(* CoDeSys 2.3 library: TcBACnet.lib *)
(* Libraries: standard.lib 5.6.98 12:03:02, TcBase.lib 14.5.09 12:14:08, TcSystem.lib 27.2.12 15:08:36, TcUtilities.lib 2.3.12 19:25:40 *)

(* Global variable list: BACnet_Globals *)
VAR_GLOBAL
(* global linkable BACnet adapter *)
	fbBACnet_Adapter	: FB_BACnet_Adapter;
(* global visible BACnet adapter reference *)
	pBACnet_Adapter		: POINTER TO FB_BACnet_Adapter;
END_VAR
VAR_GLOBAL CONSTANT
	tBACnet_ADSTimeOut		: TIME := t#5s;
END_VAR

(* Data type *)
TYPE E_BACNETACTION:
(
	BACnetAction_direct :=0,
	BACnetAction_reverse :=1
);
END_TYPE

(* Data type *)
TYPE E_BACNETADAPTERSTATUS :
(
	BACnetAdapterStatus_Init			:= 16#0,
	BACnetAdapterStatus_CheckIpAddr		:= 16#1,
	BACnetAdapterStatus_CheckParam		:= 16#2,
	BACnetAdapterStatus_GetGatewayMAC	:= 16#3,
	BACnetAdapterStatus_WaitGatewayMAC	:= 16#4,
	BACnetAdapterStatus_Complete		:= 16#8
);
END_TYPE

(* Data type *)
TYPE E_BACNETBINARYPV:
(
	BACnetBinaryPV_inactive :=0,
	BACnetBinaryPV_active :=1,
	BACnetBinaryPV_NULL := 2
);
END_TYPE

(* Data type *)
TYPE E_BACNETDATATYPES:
(
	BACnetDataType_Null :=0,
	BACnetDataType_Bool :=1,
	BACnetDataType_UnsignedInteger :=2,
	BACnetDataType_SignedInteger :=3,
	BACnetDataType_Real :=4,
	BACnetDataType_Double :=5,
	BACnetDataType_OctetString :=6,
	BACnetDataType_CharacterStringExt :=7,
	BACnetDataType_BitString :=8,
	BACnetDataType_Enumerated :=9,
	BACnetDataType_Date :=10,
	BACnetDataType_Time :=11,
	BACnetDataType_ObjectIdentifier :=12,
	BACnetDataType_DateTime :=14,
	BACnetDataType_ArrayIndex :=15,
	BACnetDataType_CalendarEntry :=16,
	BACnetDataType_ObjectType :=17,
	BACnetDataType_EventTransitionBits :=18,
	BACnetDataType_ActionList :=19,
	BACnetDataType_StatusFlags :=20,
	BACnetDataType_EventState :=21,
	BACnetDataType_Reliability :=22,
	BACnetDataType_Polarity :=23,
	BACnetDataType_EngineeringUnits :=25,
	BACnetDataType_PriorityValue :=26,
	BACnetDataType_LimitEnable :=27,
	BACnetDataType_NotifyType :=29,
	BACnetDataType_TimeStamp :=30,
	BACnetDataType_DeviceObjectPropertyReference :=31,
	BACnetDataType_DeviceStatus :=32,
	BACnetDataType_ServicesSupported :=33,
	BACnetDataType_ObjectTypesSupported :=34,
	BACnetDataType_Segmentation :=35,
	BACnetDataType_VTClass :=36,
	BACnetDataType_VTSession :=37,
	BACnetDataType_SessionKey :=38,
	BACnetDataType_Recipient :=39,
	BACnetDataType_AddressBinding :=40,
	BACnetDataType_COVSubscription :=41,
	BACnetDataType_EventType :=42,
	BACnetDataType_EventParameter :=43,
	BACnetDataType_FileAccessMethod :=44,
	BACnetDataType_ReadAccessSpecification :=45,
	BACnetDataType_ReadAccessResult :=46,
	BACnetDataType_ObjectPropertyReference :=47,
	BACnetDataType_SetpointReference :=48,
	BACnetDataType_Destination :=49,
	BACnetDataType_ProgramState :=50,
	BACnetDataType_ProgramRequest :=51,
	BACnetDataType_ProgramError :=52,
	BACnetDataType_DateRange :=53,
	BACnetDataType_DailySchedule :=54,
	BACnetDataType_SpecialEvent :=55,
	BACnetDataType_ClientCOV :=56,
	BACnetDataType_LogRecord :=57,
	BACnetDataType_LifeSafetyState :=58,
	BACnetDataType_LifeSafetyMode :=59,
	BACnetDataType_SilencedState :=60,
	BACnetDataType_LifeSafetyOperation :=61,
	BACnetDataType_BinaryPV :=62,
	BACnetDataType_DaysOfWeek :=63,
	BACnetDataType_WeekNDay :=64,
	BACnetDataType_TimeValue :=65,
	BACnetDataType_Value :=66,
	BACnetDataType_Address :=67,
	BACnetDataType_PropertyIdentifier :=68,
	BACnetDataType_EnumerationValueType :=69,
	BACnetDataType_BitFieldBit :=70,
	BACnetDataType_LogDatum :=71,
	BACnetDataType_AnyType :=72,
	BACnetDataType_PresentValue :=73,
	BACnetDataType_ContextTag :=74,
	BACnetDataType_ValueChoice :=75,
	BACnetDataType_LogStatus :=76,
	BACnetDataType_RecipientProcess :=77,
	BACnetDataType_SubscribeCOVPropertyRequest :=78,
	BACnetDataType_PropertyReference :=79,
	BACnetDataType_PropertyResult :=80,
	BACnetDataType_DeviceObjectPropertyValue :=81,
	BACnetDataType_COVNotificationRequest :=82,
	BACnetDataType_EventNotificationRequest :=83,
	BACnetDataType_NotificationParameters :=84,
	BACnetDataType_Change_of_Bitstring :=85,
	BACnetDataType_Change_of_State :=86,
	BACnetDataType_Change_of_Value :=87,
	BACnetDataType_Command_failure :=88,
	BACnetDataType_Floating_limit :=89,
	BACnetDataType_Out_of_Range :=90,
	BACnetDataType_PropertyValue :=91,
	BACnetDataType_Complex_Tag :=92,
	BACnetDataType_Change_of_life_safety :=93,
	BACnetDataType_Extended :=94,
	BACnetDataType_Buffer_ready :=95,
	BACnetDataType_Unsigned_range :=96,
	BACnetDataType_PropertyResultValue :=97,
	BACnetDataType_ServiceCOVPropSubscription :=98,
	BACnetDataType_ServiceCOVSubscription :=99,
	BACnetDataType_COVNotification :=100,
	BACnetDataType_AcknowledgeAlarmRequest :=101,
	BACnetDataType_VTOpenRequest :=102,
	BACnetDataType_Prescale :=103,
	BACnetDataType_Scale :=104,
	BACnetDataType_Action :=105,
	BACnetDataType_Error :=106,
	BACnetDataType_ErrorType :=107,
	BACnetDataType_ErrorClass :=108,
	BACnetDataType_ErrorCode :=109,
	BACnetDataType_RejectReason :=110,
	BACnetDataType_AbortReason :=111,
	BACnetDataType_BDTEntry :=112,
	BACnetDataType_IpEntry :=113,
	BACnetDataType_MaskEntry :=114,
	BACnetDataType_UnsignedIntegerArr :=258,
	BACnetDataType_CharacterStringExtArr :=263,
	BACnetDataType_ObjectIdentifierArr :=268,
	BACnetDataType_CalendarEntryArr :=272,
	BACnetDataType_ActionListArr :=275,
	BACnetDataType_PriorityValueArr :=282,
	BACnetDataType_TimeStampArr :=286,
	BACnetDataType_DeviceObjectPropertyReferenceArr :=287,
	BACnetDataType_VTClassArr :=292,
	BACnetDataType_VTSessionArr :=293,
	BACnetDataType_SessionKeyArr :=294,
	BACnetDataType_RecipientArr :=295,
	BACnetDataType_AddressBindingArr :=296,
	BACnetDataType_COVSubscriptionArr :=297,
	BACnetDataType_ReadAccessSpecificationArr :=301,
	BACnetDataType_ReadAccessResultArr :=302,
	BACnetDataType_DestinationArr :=305,
	BACnetDataType_SpecialEventArr :=311,
	BACnetDataType_LogRecordArr :=313,
	BACnetDataType_LifeSafetyStateArr :=314,
	BACnetDataType_TimeValueArr :=321,
	BACnetDataType_UnsignedIntegerList :=514,
	BACnetDataType_CharacterStringExtList :=519,
	BACnetDataType_ReadAccessSpecificationList :=557,
	BACnetDataType_ReadAccessResultList :=558,
	BACnetDataType_SpecialEventList :=567,
	BACnetDataType_LogRecordList :=569,
	BACnetDataType_TimeValueList :=577,
	BACnetDataType_ValueList :=578,
	BACnetDataType_LogDatumList :=583,
	BACnetDataType_PropertyReferenceList :=591,
	BACnetDataType_PropertyResultList :=592,
	BACnetDataType_COVNotificationRequestList :=594,
	BACnetDataType_EventNotificationRequestList :=595,
	BACnetDataType_PropertyValueList :=603,
	BACnetDataType_DailyScheduleList :=1089
);
END_TYPE

(* Data type *)
TYPE E_BACNETDEVICESTATUS:
(
	BACnetDeviceStatus_Operational :=0,
	BACnetDeviceStatus_OperationalReadOnly :=1,
	BACnetDeviceStatus_DownloadRequired :=2,
	BACnetDeviceStatus_DownloadInProgress :=3,
	BACnetDeviceStatus_NonOperational :=4,
	BACnetDeviceStatus_BackupInProgress :=5
);
END_TYPE

(* Data type *)
TYPE E_BACNETEVENTSTATE:
(
	BACnetEventState_state_normal :=0,
	BACnetEventState_fault :=1,
	BACnetEventState_offnormal :=2,
	BACnetEventState_high_limit :=3,
	BACnetEventState_low_limit :=4,
	BACnetEventState_life_safety_alarm :=5
);
END_TYPE

(* Data type *)
TYPE E_BACNETEVENTTRANSITIONBIT:
(
	BACnetEventTransitionBit_to_offnormal :=0,
	BACnetEventTransitionBit_to_fault :=1,
	BACnetEventTransitionBit_to_normal :=2
);
END_TYPE

(* Data type *)
TYPE E_BACNETEVENTTYPE:
(
	BACnetEventType_change_of_bitstring :=0,
	BACnetEventType_change_of_state :=1,
	BACnetEventType_change_of_value :=2,
	BACnetEventType_command_failure :=3,
	BACnetEventType_floating_limit :=4,
	BACnetEventType_out_of_range :=5,
	BACnetEventType_complex_event_type :=6,
	BACnetEventType_deprecated :=7,
	BACnetEventType_change_of_life_safety :=8,
	BACnetEventType_enumeration :=9,
	BACnetEventType_buffer_ready :=10,
	BACnetEventType_unsigned_range :=11
);
END_TYPE

(* Data type *)
TYPE E_BACNETFILEACCESSMETHOD:
(
	BACnetFileAccessMethod_record_access :=0,
	BACnetFileAccessMethod_stream_access :=1
);
END_TYPE

(* Data type *)
TYPE E_BACNETLIFESAFETYMODE:
(
	BACnetLifeSafetyMode_off :=0,
	BACnetLifeSafetyMode_on :=1,
	BACnetLifeSafetyMode_test :=2,
	BACnetLifeSafetyMode_manned :=3,
	BACnetLifeSafetyMode_unmanned :=4,
	BACnetLifeSafetyMode_armed :=5,
	BACnetLifeSafetyMode_disarmed :=6,
	BACnetLifeSafetyMode_prearmed :=7,
	BACnetLifeSafetyMode_slow :=8,
	BACnetLifeSafetyMode_fast :=9,
	BACnetLifeSafetyMode_disconnected :=10,
	BACnetLifeSafetyMode_enabled :=11,
	BACnetLifeSafetyMode_disabled :=12,
	BACnetLifeSafetyMode_automatic_release_disabled :=13,
	BACnetLifeSafetyMode_mode_default :=14
);
END_TYPE

(* Data type *)
TYPE E_BACNETLIFESAFETYOPERATION:
(
	BACnetLifeSafetyOperation_none :=0,
	BACnetLifeSafetyOperation_silence :=1,
	BACnetLifeSafetyOperation_silence_audible :=2,
	BACnetLifeSafetyOperation_silence_visual :=3,
	BACnetLifeSafetyOperation_reset :=4,
	BACnetLifeSafetyOperation_reset_alarm :=5,
	BACnetLifeSafetyOperation_reset_fault :=6
);
END_TYPE

(* Data type *)
TYPE E_BACNETLIMITENABLEBITS:
(
	BACnetLimitEnableBits_lowLimit :=0,
	BACnetLimitEnableBits_highLimit :=1
);
END_TYPE

(* Data type *)
TYPE E_BACNETNOTIFYTYPE:
(
	BACnetNotifyType_alarm :=0,
	BACnetNotifyType_notify_event :=1,
	BACnetNotifyType_ack_notification :=2
);
END_TYPE

(* Data type *)
TYPE E_BACNETOBJECTSUPPORTEDBITS:
(
	BACnetObjectSupportedBits_AnalogInput :=0,
	BACnetObjectSupportedBits_AnalogOutput :=1,
	BACnetObjectSupportedBits_AnalogValue :=2,
	BACnetObjectSupportedBits_BinaryInput :=3,
	BACnetObjectSupportedBits_BinaryOutput :=4,
	BACnetObjectSupportedBits_BinaryValue :=5,
	BACnetObjectSupportedBits_Calendar :=6,
	BACnetObjectSupportedBits_Command :=7,
	BACnetObjectSupportedBits_Device :=8,
	BACnetObjectSupportedBits_EventEnrollment :=9,
	BACnetObjectSupportedBits_File :=10,
	BACnetObjectSupportedBits_Group :=11,
	BACnetObjectSupportedBits_Loop :=12,
	BACnetObjectSupportedBits_MultiStateInput :=13,
	BACnetObjectSupportedBits_MultiStateOutput :=14,
	BACnetObjectSupportedBits_NotificationClass :=15,
	BACnetObjectSupportedBits_Program :=16,
	BACnetObjectSupportedBits_Schedule :=17,
	BACnetObjectSupportedBits_Averaging :=18,
	BACnetObjectSupportedBits_MultiStateValue :=19,
	BACnetObjectSupportedBits_TrendLog :=20,
	BACnetObjectSupportedBits_LifeSafetyPoint :=21,
	BACnetObjectSupportedBits_LifeSafetyZone :=22
);
END_TYPE

(* Data type *)
TYPE E_BACNETOBJECTTYPE:
(
	BACnetObjectType_AnalogInput :=0,
	BACnetObjectType_AnalogOutput :=1,
	BACnetObjectType_AnalogValue :=2,
	BACnetObjectType_BinaryInput :=3,
	BACnetObjectType_BinaryOutput :=4,
	BACnetObjectType_BinaryValue :=5,
	BACnetObjectType_Calendar :=6,
	BACnetObjectType_Command :=7,
	BACnetObjectType_Device :=8,
	BACnetObjectType_EventEnrollment :=9,
	BACnetObjectType_File :=10,
	BACnetObjectType_Group :=11,
	BACnetObjectType_Loop :=12,
	BACnetObjectType_MultiStateInput :=13,
	BACnetObjectType_MultiStateOutput :=14,
	BACnetObjectType_NotificationClass :=15,
	BACnetObjectType_Program :=16,
	BACnetObjectType_Schedule :=17,
	BACnetObjectType_Averaging :=18,
	BACnetObjectType_MultiStateValue :=19,
	BACnetObjectType_TrendLog :=20,
	BACnetObjectType_LifeSafetyPoint :=21,
	BACnetObjectType_LifeSafetyZone :=22,
	BACnetObjectType_Accumulator :=23,
	BACnetObjectType_PulseConverter :=24,

	(* keep at the end of list! *)
	BACnetObjectType_ZCount
);
END_TYPE

(* Data type *)
TYPE E_BACNETPOLARITY:
(
	BACnetPolarity_normal :=0,
	BACnetPolarity_reverse :=1
);
END_TYPE

(* Data type *)
TYPE E_BACNETPRIORITY:
(
	BACnetPriority_None :=0,
	BACnetPriority_1 :=1,
	BACnetPriority_2 :=2,
	BACnetPriority_3 :=3,
	BACnetPriority_4 :=4,
	BACnetPriority_5 :=5,
	BACnetPriority_6 :=6,
	BACnetPriority_7 :=7,
	BACnetPriority_8 :=8,
	BACnetPriority_9 :=9,
	BACnetPriority_10 :=10,
	BACnetPriority_11 :=11,
	BACnetPriority_12 :=12,
	BACnetPriority_13 :=13,
	BACnetPriority_14 :=14,
	BACnetPriority_15 :=15,
	BACnetPriority_16 :=16
);
END_TYPE

(* Data type *)
TYPE E_BACNETPROGRAMERROR:
(
	BACnetProgramError_program_normal :=0,
	BACnetProgramError_load_failed :=1,
	BACnetProgramError_progerror_internal :=2,
	BACnetProgramError_program :=3,
	BACnetProgramError_other :=4
);
END_TYPE

(* Data type *)
TYPE E_BACNETPROGRAMREQUEST:
(
	BACnetProgramRequest_ready :=0,
	BACnetProgramRequest_load :=1,
	BACnetProgramRequest_run :=2,
	BACnetProgramRequest_halt :=3,
	BACnetProgramRequest_restart :=4,
	BACnetProgramRequest_unload :=5
);
END_TYPE

(* Data type *)
TYPE E_BACNETPROGRAMSTATE:
(
	BACnetProgramState_idle :=0,
	BACnetProgramState_loading :=1,
	BACnetProgramState_running :=2,
	BACnetProgramState_waiting :=3,
	BACnetProgramState_halted :=4,
	BACnetProgramState_unloading :=5
);
END_TYPE

(* Data type *)
TYPE E_BACNETPROPERTYIDENTIFIER:
(
	BACnetPropertyIdentifier_AckedTransitions :=0,
	BACnetPropertyIdentifier_AckRequired :=1,
	BACnetPropertyIdentifier_Action :=2,
	BACnetPropertyIdentifier_ActionText :=3,
	BACnetPropertyIdentifier_ActiveText :=4,
	BACnetPropertyIdentifier_ActiveVtSessions :=5,
	BACnetPropertyIdentifier_AlarmValue :=6,
	BACnetPropertyIdentifier_AlarmValues :=7,
	BACnetPropertyIdentifier_All :=8,
	BACnetPropertyIdentifier_AllWritesSuccessful :=9,
	BACnetPropertyIdentifier_ApduSegmentTimeout :=10,
	BACnetPropertyIdentifier_ApduTimeout :=11,
	BACnetPropertyIdentifier_ApplicationSoftwareVersion :=12,
	BACnetPropertyIdentifier_Archive :=13,
	BACnetPropertyIdentifier_Bias :=14,
	BACnetPropertyIdentifier_ChangeOfStateCount :=15,
	BACnetPropertyIdentifier_ChangeOfStateTime :=16,
	BACnetPropertyIdentifier_NotificationClass :=17,
	BACnetPropertyIdentifier_ControlledVariableReference :=19,
	BACnetPropertyIdentifier_ControlledVariableUnits :=20,
	BACnetPropertyIdentifier_ControlledVariableValue :=21,
	BACnetPropertyIdentifier_CovIncrement :=22,
	BACnetPropertyIdentifier_Datelist :=23,
	BACnetPropertyIdentifier_DaylightSavingsStatus :=24,
	BACnetPropertyIdentifier_Deadband :=25,
	BACnetPropertyIdentifier_DerivativeConstant :=26,
	BACnetPropertyIdentifier_DerivativeConstantUnits :=27,
	BACnetPropertyIdentifier_Description :=28,
	BACnetPropertyIdentifier_DescriptionOfHalt :=29,
	BACnetPropertyIdentifier_DeviceAddressBinding :=30,
	BACnetPropertyIdentifier_DeviceType :=31,
	BACnetPropertyIdentifier_EffectivePeriod :=32,
	BACnetPropertyIdentifier_ElapsedActiveTime :=33,
	BACnetPropertyIdentifier_ErrorLimit :=34,
	BACnetPropertyIdentifier_EventEnable :=35,
	BACnetPropertyIdentifier_EventState :=36,
	BACnetPropertyIdentifier_EventType :=37,
	BACnetPropertyIdentifier_ExceptionSchedule :=38,
	BACnetPropertyIdentifier_FaultValues :=39,
	BACnetPropertyIdentifier_FeedbackValue :=40,
	BACnetPropertyIdentifier_FileAccessMethod :=41,
	BACnetPropertyIdentifier_FileSize :=42,
	BACnetPropertyIdentifier_FileType :=43,
	BACnetPropertyIdentifier_FirmwareRevision :=44,
	BACnetPropertyIdentifier_HighLimit :=45,
	BACnetPropertyIdentifier_InactiveText :=46,
	BACnetPropertyIdentifier_InProcess :=47,
	BACnetPropertyIdentifier_InstanceOf :=48,
	BACnetPropertyIdentifier_IntegralConstant :=49,
	BACnetPropertyIdentifier_IntegralConstantUnits :=50,
	BACnetPropertyIdentifier_IssueConfirmedNotifications :=51,
	BACnetPropertyIdentifier_LimitEnable :=52,
	BACnetPropertyIdentifier_ListOfGroupMembers :=53,
	BACnetPropertyIdentifier_ListOfObjectPropertyReferences :=54,
	BACnetPropertyIdentifier_ListOfSessionKeys :=55,
	BACnetPropertyIdentifier_LocalDate :=56,
	BACnetPropertyIdentifier_LocalTime :=57,
	BACnetPropertyIdentifier_Location :=58,
	BACnetPropertyIdentifier_LowLimit :=59,
	BACnetPropertyIdentifier_ManipulatedVariableReference :=60,
	BACnetPropertyIdentifier_MaximumOutput :=61,
	BACnetPropertyIdentifier_MaxApduLengthAccepted :=62,
	BACnetPropertyIdentifier_MaxInfoFrames :=63,
	BACnetPropertyIdentifier_MaxMaster :=64,
	BACnetPropertyIdentifier_MaxPresValue :=65,
	BACnetPropertyIdentifier_MinimumOfftime :=66,
	BACnetPropertyIdentifier_MinimumOntime :=67,
	BACnetPropertyIdentifier_MinimumOutput :=68,
	BACnetPropertyIdentifier_MinPresValue :=69,
	BACnetPropertyIdentifier_ModelName :=70,
	BACnetPropertyIdentifier_ModificationDate :=71,
	BACnetPropertyIdentifier_NotifyType :=72,
	BACnetPropertyIdentifier_NumberOfAPDURetries :=73,
	BACnetPropertyIdentifier_NumberOfStates :=74,
	BACnetPropertyIdentifier_ObjectIdentifier :=75,
	BACnetPropertyIdentifier_ObjectList :=76,
	BACnetPropertyIdentifier_ObjectName :=77,
	BACnetPropertyIdentifier_ObjectReference :=78,
	BACnetPropertyIdentifier_ObjectType :=79,
	BACnetPropertyIdentifier_Optional :=80,
	BACnetPropertyIdentifier_OutOfService :=81,
	BACnetPropertyIdentifier_OutputUnits :=82,
	BACnetPropertyIdentifier_EventParameters :=83,
	BACnetPropertyIdentifier_Polarity :=84,
	BACnetPropertyIdentifier_PresentValue :=85,
	BACnetPropertyIdentifier_Priority :=86,
	BACnetPropertyIdentifier_PriorityArray :=87,
	BACnetPropertyIdentifier_PriorityForWriting :=88,
	BACnetPropertyIdentifier_ProcessIdentifier :=89,
	BACnetPropertyIdentifier_ProgramChange :=90,
	BACnetPropertyIdentifier_ProgramLocation :=91,
	BACnetPropertyIdentifier_ProgramState :=92,
	BACnetPropertyIdentifier_ProportionalConstant :=93,
	BACnetPropertyIdentifier_ProportionalConstantUnits :=94,
	BACnetPropertyIdentifier_ProtocolObjectTypesSupported :=96,
	BACnetPropertyIdentifier_ProtocolServicesSupported :=97,
	BACnetPropertyIdentifier_ProtocolVersion :=98,
	BACnetPropertyIdentifier_ReadOnly :=99,
	BACnetPropertyIdentifier_ReasonForHalt :=100,
	BACnetPropertyIdentifier_Recipient :=101,
	BACnetPropertyIdentifier_RecipientList :=102,
	BACnetPropertyIdentifier_Reliability :=103,
	BACnetPropertyIdentifier_RelinquishDefault :=104,
	BACnetPropertyIdentifier_Required :=105,
	BACnetPropertyIdentifier_Resolution :=106,
	BACnetPropertyIdentifier_SegmentationSupported :=107,
	BACnetPropertyIdentifier_Setpoint :=108,
	BACnetPropertyIdentifier_SetpointReference :=109,
	BACnetPropertyIdentifier_StateText :=110,
	BACnetPropertyIdentifier_StatusFlags :=111,
	BACnetPropertyIdentifier_SystemStatus :=112,
	BACnetPropertyIdentifier_TimeDelay :=113,
	BACnetPropertyIdentifier_TimeOfActiveTimeReset :=114,
	BACnetPropertyIdentifier_TimeOfStateCountReset :=115,
	BACnetPropertyIdentifier_TimeSynchronizationRecipients :=116,
	BACnetPropertyIdentifier_Units :=117,
	BACnetPropertyIdentifier_UpdateInterval :=118,
	BACnetPropertyIdentifier_UtcOffset :=119,
	BACnetPropertyIdentifier_VendorIdentifier :=120,
	BACnetPropertyIdentifier_VendorName :=121,
	BACnetPropertyIdentifier_VtClassesSupported :=122,
	BACnetPropertyIdentifier_WeeklySchedule :=123,
	BACnetPropertyIdentifier_AttemptedSamples :=124,
	BACnetPropertyIdentifier_AverageValue :=125,
	BACnetPropertyIdentifier_BufferSize :=126,
	BACnetPropertyIdentifier_ClientCovIncrement :=127,
	BACnetPropertyIdentifier_CovResubscriptionInterval :=128,
	BACnetPropertyIdentifier_EventTimeStamps :=130,
	BACnetPropertyIdentifier_LogBuffer :=131,
	BACnetPropertyIdentifier_LogDeviceObjectProperty :=132,
	BACnetPropertyIdentifier_LogEnable :=133,
	BACnetPropertyIdentifier_LogInterval :=134,
	BACnetPropertyIdentifier_MaximumValue :=135,
	BACnetPropertyIdentifier_MinimumValue :=136,
	BACnetPropertyIdentifier_NotificationThreshold :=137,
	BACnetPropertyIdentifier_ProtocolRevision :=139,
	BACnetPropertyIdentifier_RecordsSinceNotification :=140,
	BACnetPropertyIdentifier_RecordCount :=141,
	BACnetPropertyIdentifier_StartTime :=142,
	BACnetPropertyIdentifier_StopTime :=143,
	BACnetPropertyIdentifier_StopWhenFull :=144,
	BACnetPropertyIdentifier_TotalRecordCount :=145,
	BACnetPropertyIdentifier_ValidSamples :=146,
	BACnetPropertyIdentifier_WindowInterval :=147,
	BACnetPropertyIdentifier_WindowSamples :=148,
	BACnetPropertyIdentifier_MaximumValueTimestamp :=149,
	BACnetPropertyIdentifier_MinimumValueTimestamp :=150,
	BACnetPropertyIdentifier_VarianceValue :=151,
	BACnetPropertyIdentifier_ActiveCovSubscriptions :=152,
	BACnetPropertyIdentifier_BackupFailureTimeout :=153,
	BACnetPropertyIdentifier_ConfigurationFiles :=154,
	BACnetPropertyIdentifier_DatabaseRevision :=155,
	BACnetPropertyIdentifier_DirectReading :=156,
	BACnetPropertyIdentifier_LastRestoreTime :=157,
	BACnetPropertyIdentifier_MaintenanceRequired :=158,
	BACnetPropertyIdentifier_MemberOf :=159,
	BACnetPropertyIdentifier_Mode :=160,
	BACnetPropertyIdentifier_OperationExpected :=161,
	BACnetPropertyIdentifier_Setting :=162,
	BACnetPropertyIdentifier_Silenced :=163,
	BACnetPropertyIdentifier_TrackingValue :=164,
	BACnetPropertyIdentifier_ZoneMembers :=165,
	BACnetPropertyIdentifier_LifeSafetyAlarmValues :=166,
	BACnetPropertyIdentifier_MaxSegmentsAccepted :=167,
	BACnetPropertyIdentifier_ProfileName :=168,
	BACnetPropertyIdentifier_InternalUse :=169,
	BACnetPropertyIdentifier_LastNotifyRecord :=173,
	BACnetPropertyIdentifier_ScheduleDefault :=174,
	BACnetPropertyIdentifier_AcceptedModes :=175,
	BACnetPropertyIdentifier_AdjustValue :=176,
	BACnetPropertyIdentifier_Count :=177,
	BACnetPropertyIdentifier_CountBeforeChange :=178,
	BACnetPropertyIdentifier_CovPeriod :=180,
	BACnetPropertyIdentifier_InputReference :=181,
	BACnetPropertyIdentifier_LimitMonitoringInverval :=182,
	BACnetPropertyIdentifier_LoggingObject :=183,
	BACnetPropertyIdentifier_LoggingRecord :=184,
	BACnetPropertyIdentifier_Prescale :=185,
	BACnetPropertyIdentifier_PulseRate :=186,
	BACnetPropertyIdentifier_Scale :=187,
	BACnetPropertyIdentifier_ScaleFactor :=188,
	BACnetPropertyIdentifier_UpdateTime :=189,
	BACnetPropertyIdentifier_ValueBeforeChange :=190,
	BACnetPropertyIdentifier_ValueSet :=191,
	BACnetPropertyIdentifier_ValueChangeTime :=192
);
END_TYPE

(* Data type *)
TYPE E_BACNETRELIABILITY:
(
	BACnetReliability_no_fault_detected :=0,
	BACnetReliability_no_sensor :=1,
	BACnetReliability_over_range :=2,
	BACnetReliability_under_range :=3,
	BACnetReliability_open_loop :=4,
	BACnetReliability_shorted_loop :=5,
	BACnetReliability_no_output :=6,
	BACnetReliability_unreliable_other :=7,
	BACnetReliability_process_error :=8,
	BACnetReliability_multi_state_fault :=9,
	BACnetReliability_configuration_error :=10,
	BACnetReliability_member_fault :=11,
	BACnetReliability_communication_error :=12
);
END_TYPE

(* Data type *)
TYPE E_BACNETSEGMENTATION:
(
	BACnetSegmentation_both :=0,
	BACnetSegmentation_transmit :=1,
	BACnetSegmentation_receive :=2,
	BACnetSegmentation_no :=3
);
END_TYPE

(* Data type *)
TYPE E_BACNETSERVICESUPPORTEDBITS:
(
	BACnetServiceSupportedBits_AcknowledgeAlarm :=0,
	BACnetServiceSupportedBits_ConfirmedCOVNotification :=1,
	BACnetServiceSupportedBits_ConfirmedEventNotification :=2,
	BACnetServiceSupportedBits_GetAlarmSummary :=3,
	BACnetServiceSupportedBits_GetEnrollmentSummary :=4,
	BACnetServiceSupportedBits_SubscribeCOV :=5,
	BACnetServiceSupportedBits_AtomicReadFile :=6,
	BACnetServiceSupportedBits_AtomicWriteFile :=7,
	BACnetServiceSupportedBits_AddListElement :=8,
	BACnetServiceSupportedBits_RemoveListElement :=9,
	BACnetServiceSupportedBits_CreateObject :=10,
	BACnetServiceSupportedBits_DeleteObject :=11,
	BACnetServiceSupportedBits_ReadProperty :=12,
	BACnetServiceSupportedBits_ReadPropertyConditional :=13,
	BACnetServiceSupportedBits_ReadPropertyMultiple :=14,
	BACnetServiceSupportedBits_WriteProperty :=15,
	BACnetServiceSupportedBits_WritePropertyMultiple :=16,
	BACnetServiceSupportedBits_DeviceCommunicationControl :=17,
	BACnetServiceSupportedBits_ConfirmedPrivateTransfer :=18,
	BACnetServiceSupportedBits_ConfirmedTextMessage :=19,
	BACnetServiceSupportedBits_ReinitializeDevice :=20,
	BACnetServiceSupportedBits_VtOpen :=21,
	BACnetServiceSupportedBits_VtClose :=22,
	BACnetServiceSupportedBits_VtData :=23,
	BACnetServiceSupportedBits_Authenticate :=24,
	BACnetServiceSupportedBits_RequestKey :=25,
	BACnetServiceSupportedBits_IAm :=26,
	BACnetServiceSupportedBits_IHave :=27,
	BACnetServiceSupportedBits_UnconfirmedCOVNotification :=28,
	BACnetServiceSupportedBits_UnconfirmedEventNotification :=29,
	BACnetServiceSupportedBits_UnconfirmedPrivateTransfer :=30,
	BACnetServiceSupportedBits_UnconfirmedTextMessage :=31,
	BACnetServiceSupportedBits_TimeSynchronization :=32,
	BACnetServiceSupportedBits_WhoHas :=33,
	BACnetServiceSupportedBits_WhoIs :=34,
	BACnetServiceSupportedBits_ReadRange :=35,
	BACnetServiceSupportedBits_UtcTimeSynchronization :=36,
	BACnetServiceSupportedBits_LifeSafetyOperation :=37,
	BACnetServiceSupportedBits_SubscribeCOVProperty :=38,
	BACnetServiceSupportedBits_GetEventInformation :=39
);
END_TYPE

(* Data type *)
TYPE E_BACNETSILENCEDSTATE:
(
	BACnetSilencedState_unsilenced :=0,
	BACnetSilencedState_audible_silenced :=1,
	BACnetSilencedState_visible_silenced :=2,
	BACnetSilencedState_all_silenced :=3
);
END_TYPE

(* Data type *)
TYPE E_BACNETSTATUSFLAGS:
(
	BACnetStatusFlags_in_alarm :=0,
	BACnetStatusFlags_fault :=1,
	BACnetStatusFlags_overridden :=2,
	BACnetStatusFlags_out_of_service :=3
);
END_TYPE

(* Data type *)
TYPE E_BACNETUNIT:
(
	BACnetUnit_Area_square_meters :=0,
	BACnetUnit_Area_square_feet :=1,
	BACnetUnit_Electrical_milliamperes :=2,
	BACnetUnit_Electrical_amperes :=3,
	BACnetUnit_Electrical_ohms :=4,
	BACnetUnit_Electrical_volts :=5,
	BACnetUnit_Electrical_kilovolts :=6,
	BACnetUnit_Electrical_megavolts :=7,
	BACnetUnit_Electrical_volt_amperes :=8,
	BACnetUnit_Electrical_kilovolt_amperes :=9,
	BACnetUnit_Electrical_megavolt_amperes :=10,
	BACnetUnit_Electrical_volt_amperes_reactive :=11,
	BACnetUnit_Electrical_kilovolt_amperes_reactive :=12,
	BACnetUnit_Electrical_megavolt_amperes_reactive :=13,
	BACnetUnit_Electrical_degrees_phase :=14,
	BACnetUnit_Electrical_power_factor :=15,
	BACnetUnit_Energy_joules :=16,
	BACnetUnit_Energy_kilojoules :=17,
	BACnetUnit_Energy_watt_hours :=18,
	BACnetUnit_Energy_kilowatt_hours :=19,
	BACnetUnit_Energy_btus :=20,
	BACnetUnit_Energy_therms :=21,
	BACnetUnit_Energy_ton_hours :=22,
	BACnetUnit_Enthalpy_joules_per_kilogram_dry_air :=23,
	BACnetUnit_Enthalpy_btus_per_pound_dry_air :=24,
	BACnetUnit_Frequency_cycles_per_hour :=25,
	BACnetUnit_Frequency_cycles_per_minute :=26,
	BACnetUnit_Frequency_hertz :=27,
	BACnetUnit_Humidity_grams_of_water_per_kilogram_dry_air :=28,
	BACnetUnit_Humidity_percent_relative_humidity :=29,
	BACnetUnit_Length_millimeters :=30,
	BACnetUnit_Length_meters :=31,
	BACnetUnit_Length_inches :=32,
	BACnetUnit_Length_feet :=33,
	BACnetUnit_Light_watts_per_square_foot :=34,
	BACnetUnit_Light_watts_per_square_meter :=35,
	BACnetUnit_Light_lumens :=36,
	BACnetUnit_Light_luxes :=37,
	BACnetUnit_Light_foot_candles :=38,
	BACnetUnit_Mass_kilograms :=39,
	BACnetUnit_Mass_pounds_mass :=40,
	BACnetUnit_Mass_tons :=41,
	BACnetUnit_Mass_Flow_kilograms_per_second :=42,
	BACnetUnit_Mass_Flow_kilograms_per_minute :=43,
	BACnetUnit_Mass_Flow_kilograms_per_hour :=44,
	BACnetUnit_Mass_Flow_pounds_mass_per_minute :=45,
	BACnetUnit_Mass_Flow_pounds_mass_per_hour :=46,
	BACnetUnit_Power_watts :=47,
	BACnetUnit_Power_kilowatts :=48,
	BACnetUnit_Power_megawatts :=49,
	BACnetUnit_Power_btus_per_hour :=50,
	BACnetUnit_Power_horsepower :=51,
	BACnetUnit_Power_tons_refrigeration :=52,
	BACnetUnit_Pressure_pascals :=53,
	BACnetUnit_Pressure_kilopascals :=54,
	BACnetUnit_Pressure_bars :=55,
	BACnetUnit_Pressure_pounds_force_per_square_inch :=56,
	BACnetUnit_Pressure_centimeters_of_water :=57,
	BACnetUnit_Pressure_inches_of_water :=58,
	BACnetUnit_Pressure_millimeters_of_mercury :=59,
	BACnetUnit_Pressure_centimeters_of_mercury :=60,
	BACnetUnit_Pressure_inches_of_mercury :=61,
	BACnetUnit_Temperature_degrees_Celsius :=62,
	BACnetUnit_Temperature_degrees_Kelvin :=63,
	BACnetUnit_Temperature_degrees_Fahrenheit :=64,
	BACnetUnit_Temperature_degree_days_Celsius :=65,
	BACnetUnit_Temperature_degree_days_Fahrenheit :=66,
	BACnetUnit_Time_years :=67,
	BACnetUnit_Time_months :=68,
	BACnetUnit_Time_weeks :=69,
	BACnetUnit_Time_days :=70,
	BACnetUnit_Time_hours :=71,
	BACnetUnit_Time_minutes :=72,
	BACnetUnit_Time_seconds :=73,
	BACnetUnit_Velocity_meters_per_second :=74,
	BACnetUnit_Velocity_kilometers_per_hour :=75,
	BACnetUnit_Velocity_feet_per_second :=76,
	BACnetUnit_Velocity_feet_per_minute :=77,
	BACnetUnit_Velocity_miles_per_hour :=78,
	BACnetUnit_Volume_cubic_feet :=79,
	BACnetUnit_Volume_cubic_meters :=80,
	BACnetUnit_Volume_imperial_gallons :=81,
	BACnetUnit_Volume_liters :=82,
	BACnetUnit_Volume_us_gallons :=83,
	BACnetUnit_VolumeFlow_cubic_feet_per_minute :=84,
	BACnetUnit_VolumeFlow_cubic_meters_per_second :=85,
	BACnetUnit_VolumeFlow_imperial_gallons_per_minute :=86,
	BACnetUnit_VolumeFlow_liters_per_second :=87,
	BACnetUnit_VolumeFlow_liters_per_minute :=88,
	BACnetUnit_VolumeFlow_us_gallons_per_minute :=89,
	BACnetUnit_Other_degrees_angular :=90,
	BACnetUnit_Other_degrees_Celsius_per_hour :=91,
	BACnetUnit_Other_degrees_Celsius_per_minute :=92,
	BACnetUnit_Other_degrees_Fahrenheit_per_hour :=93,
	BACnetUnit_Other_degrees_Fahrenheit_per_minute :=94,
	BACnetUnit_Other_no_units :=95,
	BACnetUnit_Other_parts_per_million :=96,
	BACnetUnit_Other_parts_per_billion :=97,
	BACnetUnit_Other_percent :=98,
	BACnetUnit_Other_percent_per_second :=99,
	BACnetUnit_Other_per_minute :=100,
	BACnetUnit_Other_per_second :=101,
	BACnetUnit_Other_psi_per_degree_Fahrenheit :=102,
	BACnetUnit_Other_radians :=103,
	BACnetUnit_Other_revolutions_per_minute :=104,
	BACnetUnit_Currency_currency1 :=105,
	BACnetUnit_Currency_currency2 :=106,
	BACnetUnit_Currency_currency3 :=107,
	BACnetUnit_Currency_currency4 :=108,
	BACnetUnit_Currency_currency5 :=109,
	BACnetUnit_Currency_currency6 :=110,
	BACnetUnit_Currency_currency7 :=111,
	BACnetUnit_Currency_currency8 :=112,
	BACnetUnit_Currency_currency9 :=113,
	BACnetUnit_Currency_currency10 :=114,
	BACnetUnit_Area_square_inches :=115,
	BACnetUnit_Area_square_centimeters :=116,
	BACnetUnit_Enthalpy_btus_per_pound :=117,
	BACnetUnit_Length_centimeters :=118,
	BACnetUnit_Mass_Flow_pounds_mass_per_second :=119,
	BACnetUnit_Temperature_delta_degrees_Fahrenheit :=120,
	BACnetUnit_Temperature_delta_degrees_Kelvin :=121,
	BACnetUnit_Electrical_kilohms :=122,
	BACnetUnit_Electrical_megohms :=123,
	BACnetUnit_Electrical_millivolts :=124,
	BACnetUnit_Energy_kilojoules_per_kilogram :=125,
	BACnetUnit_Energy_megajoules :=126,
	BACnetUnit_Entropy_joules_per_degree_Kelvin :=127,
	BACnetUnit_Entropy_joules_per_kilogram_degree_Kelvin :=128,
	BACnetUnit_Frequency_kilohertz :=129,
	BACnetUnit_Frequency_megahertz :=130,
	BACnetUnit_Frequency_per_hour :=131,
	BACnetUnit_Power_milliwatts :=132,
	BACnetUnit_Pressure_hectopascals :=133,
	BACnetUnit_Pressure_millibars :=134,
	BACnetUnit_VolumeFlow_cubic_meters_per_hour :=135,
	BACnetUnit_VolumeFlow_liters_per_hour :=136,
	BACnetUnit_Other_kilowatt_hours_per_square_meter :=137,
	BACnetUnit_Other_kilowatt_hours_per_square_foot :=138,
	BACnetUnit_Other_megajoules_per_square_meter :=139,
	BACnetUnit_Other_megajoules_per_square_foot :=140,
	BACnetUnit_Other_watts_per_square_meter_degree_kelvin :=141,
	BACnetUnit_VolumeFlow_cubic_feet_per_second :=142,
	BACnetUnit_Other_percent_obscuration_per_foot :=143,
	BACnetUnit_Other_percent_obscuration_per_meter :=144
);
END_TYPE

(* Data type *)
TYPE ST_BACnet_ConfirmedServiceDiag :
STRUCT
	nReqSend: DWORD; (* ULONG *)
	nReqSendFail: DWORD; (* ULONG *)
	nReqRecv: DWORD; (* ULONG *)
	nReqRecvFail: DWORD; (* ULONG *)
	nAckSend: DWORD; (* ULONG *)
	nAckSendFail: DWORD; (* ULONG *)
	nAckRecv: DWORD; (* ULONG *)
	nAckRecvFail: DWORD; (* ULONG *)
END_STRUCT
END_TYPE

(* Data type *)
TYPE ST_BACnet_Date :
STRUCT
	nYear		: BYTE; (* year minus 1900 X'FF' = unspecified *)
	nMonth		: BYTE; (* (1.. 12) 1 = January X'FF' = unspecified *)
	nDay		: BYTE;	(* day OF month (1..31), X'FF' = unspecified *)
	nDayOfWeek	: BYTE;	(* day OF week (1..7) 1 = Monday -- 7 = Sunday -- X'FF' = unspecified *)
END_STRUCT
END_TYPE

(* Data type *)
TYPE ST_BACnet_DateTime :
STRUCT
	stDate		: ST_BACnet_Date;
	stTime		: ST_BACnet_Time;
END_STRUCT
END_TYPE

(* Data type *)
TYPE ST_BACnet_DiagEthStatistics :
STRUCT
	ethStat: ST_BACnet_TcIoEthStatistic;
	txRxErrCnt: ST_BACnet_TcIoEthTxRxErrorCount;
END_STRUCT
END_TYPE

(* Data type *)
TYPE ST_BACnet_Diagnosis :
STRUCT
	ethDevice: ST_BACnet_DiagEthStatistics;
	execTiming: ST_BACnet_DiagnosisTiming;
	frameStatistics: ST_BACnet_FrameStatistics;
	nRes1 : DWORD;
	info: ST_BACnet_Info;
	nRes2 : DWORD;
	serverInfo: ST_BACnet_ServerStatistics;
	lastUpdate: ST_BACnet_DateTime;
	nRes3 : DWORD;
END_STRUCT
END_TYPE

(* Data type *)
TYPE ST_BACnet_DiagnosisTiming :
STRUCT
	msIoInCurExecutionTime: DWORD; (* ULONG *)
	msIoInMinExecutionTime: DWORD; (* ULONG *)
	msIoInMaxExecutionTime: DWORD; (* ULONG *)
	msIoOutCurExecutionTime: DWORD; (* ULONG *)
	msIoOutMinExecutionTime: DWORD; (* ULONG *)
	msIoOutMaxExecutionTime: DWORD; (* ULONG *)
	msCycleCurExecutionTime: DWORD; (* ULONG *)
	msCycleMinExecutionTime: DWORD; (* ULONG *)
	msCycleMaxExecutionTime: DWORD; (* ULONG *)
	msInputCurDistanceTime: DWORD; (* ULONG *)
	msInputMinDistanceTime: DWORD; (* ULONG *)
	msInputMaxDistanceTime: DWORD; (* ULONG *)
END_STRUCT
END_TYPE

(* Data type *)
TYPE ST_BACnet_EventTransitionBits:
STRUCT
	to_offnormal : BOOL;
	to_fault : BOOL;
	to_normal : BOOL;
END_STRUCT
END_TYPE

(* Data type *)
TYPE ST_BACnet_FrameStatistics :
STRUCT
	confirmed: ARRAY[0..29] OF ST_BACnet_ConfirmedServiceDiag; (* [SERVICE_CONFIRMED_MAX + 1]; 29 + 1 *)
	unConfirmed: ARRAY[0..9] OF ST_BACnet_UnConfirmedServiceDiag; (* [SERVICE_UNCONFIRMED_MAX + 1]; 9 *)
	nSegmSendTimeouts: DWORD; (* ULONG *)
	nFrameAllocFailCnt: DWORD; (* ULONG *)
	nFrameSendCnt: DWORD; (* ULONG *)
	nFrameSendFailCnt: DWORD; (* ULONG *)
	nFrameRecvCnt: DWORD; (* ULONG *)
	nFrameRecvFailCnt: DWORD; (* ULONG *)
	nLinkStatusChangedCnt: DWORD; (* ULONG *)
END_STRUCT
END_TYPE

(* Data type *)
TYPE ST_BACnet_Info :
STRUCT
	nAmsAllocCnt: DINT; (* LONG *)
	nAmsAllocCntMax: DWORD; (* ULONG *)
	nAmsAllocFailCnt: DWORD; (* ULONG *)
	nAvailPhysMemBytes: DWORD; (* ULONG *)
	nAvailFlashMemBytes: ARRAY[0..1] OF DWORD; (* ULONGLONG *)
	nRecvFrameFifoSize: DWORD; (* ULONG *)
	nEmptyFrameFifoSize: DWORD; (* ULONG *)
	nRecvSegmUDPFramesListSize: DWORD; (* ULONG *)
	nRecvSegmFramesListSize: DWORD; (* ULONG *)
	nSendSegmFramesListSize: DWORD; (* ULONG *)
	nClientScanListSize: DWORD; (* ULONG *)
	nAdsRequestListSize: DWORD; (* ULONG *)
END_STRUCT
END_TYPE

(* Data type *)
TYPE ST_BACnet_LimitEnable:
STRUCT
	lowLimitEnable : BOOL;
	highLimitEnable : BOOL;
END_STRUCT
END_TYPE

(* Data type *)
TYPE ST_BACnet_ObjectTypesSupported:
STRUCT
	SuppAnalogInput : BOOL;
	SuppAnalogOutput : BOOL;
	SuppAnalogValue : BOOL;
	SuppBinaryInput : BOOL;
	SuppBinaryOutput : BOOL;
	SuppBinaryValue : BOOL;
	SuppCalendar : BOOL;
	SuppCommand : BOOL;
	SuppDevice : BOOL;
	SuppEventEnrollment : BOOL;
	SuppFile : BOOL;
	SuppGroup : BOOL;
	SuppLoop : BOOL;
	SuppMultiStateInput : BOOL;
	SuppMultiStateOutput : BOOL;
	SuppNotificationClass : BOOL;
	SuppProgram : BOOL;
	SuppSchedule : BOOL;
	SuppAveraging : BOOL;
	SuppMultiStateValue : BOOL;
	SuppTrendLog : BOOL;
	SuppLifeSafetyPoint : BOOL;
	SuppLifeSafetyZone : BOOL;
END_STRUCT
END_TYPE

(* Data type *)
TYPE ST_BACnet_ProgramHandshakeRequests :
STRUCT
	bLoad	: BOOL;
	bSetup	: BOOL;
	bRun	: BOOL;
	bHalt	: BOOL;
	bUnload	: BOOL;
END_STRUCT
END_TYPE

(* Data type *)
TYPE ST_BACnet_ProgramHandshakeStates :
STRUCT
	bIdle		: BOOL;
	bLoading	: BOOL;
	bRunning	: BOOL;
	bWaiting	: BOOL;
	bHalted		: BOOL;
	bUnloading	: BOOL;
END_STRUCT
END_TYPE

(* Data type *)
TYPE ST_BACnet_ServerStatistics :
STRUCT
	nOpenRequests: DWORD; (* ULONG *)
	nRequestRetries: DWORD; (* ULONG *)
	nRequestTimeOuts: DWORD; (* ULONG *)
	nPropChanges: DWORD; (* ULONG *)
	nPersistWrites: DWORD; (* ULONG *)
	persistChangeSetId: DWORD; (* ULONG *)
	secpersistNextWrite: DWORD; (* ULONG *)
	persistLastWrite: ST_BACnet_DateTime;
END_STRUCT
END_TYPE

(* Data type *)
TYPE ST_BACnet_ServicesSupported:
STRUCT
	SuppAcknowledgeAlarm : BOOL;
	SuppConfirmedCOVNotification : BOOL;
	SuppConfirmedEventNotification : BOOL;
	SuppGetAlarmSummary : BOOL;
	SuppGetEnrollmentSummary : BOOL;
	SuppSubscribeCOV : BOOL;
	SuppAtomicReadFile : BOOL;
	SuppAtomicWriteFile : BOOL;
	SuppAddListElement : BOOL;
	SuppRemoveListElement : BOOL;
	SuppCreateObject : BOOL;
	SuppDeleteObject : BOOL;
	SuppReadProperty : BOOL;
	SuppReadPropertyConditional : BOOL;
	SuppReadPropertyMultiple : BOOL;
	SuppWriteProperty : BOOL;
	SuppWritePropertyMultiple : BOOL;
	SuppDeviceCommunicationControl : BOOL;
	SuppConfirmedPrivateTransfer : BOOL;
	SuppConfirmedTextMessage : BOOL;
	SuppReinitializeDevice : BOOL;
	SuppVtOpen : BOOL;
	SuppVtClose : BOOL;
	SuppVtData : BOOL;
	SuppAuthenticate : BOOL;
	SuppRequestKey : BOOL;
	SuppIAm : BOOL;
	SuppIHave : BOOL;
	SuppUnconfirmedCOVNotification : BOOL;
	SuppUnconfirmedEventNotification : BOOL;
	SuppUnconfirmedPrivateTransfer : BOOL;
	SuppUnconfirmedTextMessage : BOOL;
	SuppTimeSynchronization : BOOL;
	SuppWhoHas : BOOL;
	SuppWhoIs : BOOL;
	SuppReadRange : BOOL;
	SuppUtcTimeSynchronization : BOOL;
	SuppLifeSafetyOperation : BOOL;
	SuppSubscribeCOVProperty : BOOL;
	SuppGetEventInformation : BOOL;
END_STRUCT
END_TYPE

(* Data type *)
TYPE ST_BACnet_StatusFlags:
STRUCT
	in_alarm : BOOL;
	fault : BOOL;
	overridden : BOOL;
	out_of_service : BOOL;
END_STRUCT
END_TYPE

(* Data type *)
TYPE ST_BACnet_TcIoEthStatistic :
STRUCT
	dcTimeStamp: ARRAY[0..1] OF DWORD; (* ULONGLONG *)
	sendFrames: DWORD; (* ULONG *)
	recvFrames: DWORD; (* ULONG *)
	sendTimeRTime: DWORD; (* ULONG *)
	recvTimeRTime: DWORD; (* ULONG *)
	sendTimeNdis: DWORD; (* ULONG *)
	recvTimeNdis: DWORD; (* ULONG *)
END_STRUCT
END_TYPE

(* Data type *)
TYPE ST_BACnet_TcIoEthTxRxErrorCount :
STRUCT
	txCnt: DWORD; (* ULONG *)
	rxCnt: DWORD; (* ULONG *)
END_STRUCT
END_TYPE

(* Data type *)
TYPE ST_BACnet_Time :
STRUCT
	nHour		: BYTE; (* hour (0..23), (X'FF') = unspecified *)
	nMinute		: BYTE;	(* minute (0..59), (X'FF') = unspecified *)
	nSecond		: BYTE; (* (0..59), (X'FF') = unspecified *)
	nHundredths	: BYTE;	(* hundredths (0..99), (X'FF') = unspecified *)
END_STRUCT
END_TYPE

(* Data type *)
TYPE ST_BACnet_UnConfirmedServiceDiag :
STRUCT
	nReqSend: DWORD; (* ULONG *)
	nReqSendFail: DWORD; (* ULONG *)
	nReqRecv: DWORD; (* ULONG *)
	nReqRecvFail: DWORD; (* ULONG *)
END_STRUCT
END_TYPE

(* POU _F_BACnet_BitFieldBit, ST *)
FUNCTION _F_BACnet_BitFieldBit : WORD
VAR_INPUT
	Bit	:	WORD;
END_VAR
VAR
END_VAR
_F_BACnet_BitFieldBit := (Bit/8) * 8 + (bit MOD 8);
END_FUNCTION

(* POU _F_BACnet_IsBitFieldBitSet, ST *)
FUNCTION _F_BACnet_IsBitFieldBitSet : BOOL
VAR_INPUT
	data	:	DWORD;
	Bit		:	WORD;
END_VAR
VAR
END_VAR
_F_BACnet_IsBitFieldBitSet:= (data AND (SHR(DWORD#16#00008000,_F_BACnet_BitFieldBit(Bit)))) > 0;
END_FUNCTION

(* POU _F_BACnet_SetBitFieldBit, ST *)
FUNCTION _F_BACnet_SetBitFieldBit : DWORD
VAR_INPUT
	ptrData		:	POINTER TO DWORD;
	Bit			:	WORD;
END_VAR
VAR
END_VAR
ptrData^ := ptrData^ AND NOT  (SHR(DWORD#00008000,_F_BACnet_BitFieldBit(Bit)));
_F_BACnet_SetBitFieldBit := ptrData^;
END_FUNCTION

(* POU _F_BACnet_UnSetBitFieldBit, ST *)
FUNCTION _F_BACnet_UnSetBitFieldBit : DWORD
VAR_INPUT
	ptrData		:	POINTER TO DWORD;
	Bit			:	WORD;
END_VAR
VAR
END_VAR
ptrData^ := ptrData^ OR (SHR(DWORD#00008000,_F_BACnet_BitFieldBit(Bit)));
_F_BACnet_UnSetBitFieldBit := ptrData^;
END_FUNCTION

(* POU F_BACnet_EventTransitionFlags, ST *)
FUNCTION F_BACnet_EventTransitionFlags : ST_BACnet_EventTransitionBits
VAR_INPUT
	data	: WORD;
END_VAR
VAR
END_VAR
F_BACnet_EventTransitionFlags.to_normal := _F_BACnet_IsBitFieldBitSet( data:=data, Bit:=BACnetEventTransitionBit_to_normal);
F_BACnet_EventTransitionFlags.to_offnormal := _F_BACnet_IsBitFieldBitSet( data:=data, Bit:=BACnetEventTransitionBit_to_offnormal);
F_BACnet_EventTransitionFlags.to_fault := _F_BACnet_IsBitFieldBitSet( data:=data, Bit:=BACnetEventTransitionBit_to_fault);
END_FUNCTION

(* POU F_BACnet_GetObjId, ST *)
FUNCTION F_BACnet_GetObjId : DWORD
VAR_INPUT
	ObjectType		: E_BACNETOBJECTTYPE;
	ObjectInstance	: UDINT;
END_VAR
VAR
END_VAR
F_BACnet_GetObjId := F_BACnet_GetObjInstance(ObjectInstance) + SHL(INT_TO_UDINT(ObjectType), 22);
END_FUNCTION

(* POU F_BACnet_GetObjInstance, ST *)
FUNCTION F_BACnet_GetObjInstance : UDINT
VAR_INPUT
	nObjectId : DWORD;
END_VAR
VAR
END_VAR
F_BACnet_GetObjInstance := nObjectId AND 16#003FFFFF;
END_FUNCTION

(* POU F_BACnet_GetObjType, ST *)
FUNCTION F_BACnet_GetObjType : E_BACNETOBJECTTYPE
VAR_INPUT
	nObjectId : DWORD;
END_VAR
VAR
END_VAR
F_BACnet_GetObjType := DWORD_TO_WORD(SHR((nObjectId AND 16#FFC00000), 22));
END_FUNCTION

(* POU F_BACnet_IsFinite, ST *)
FUNCTION F_BACnet_IsFinite : BOOL
VAR_INPUT
	fValue		: REAL;
END_VAR
VAR
	fArg		: T_Arg;
END_VAR
fArg.cbLen := SIZEOF(fValue);
fArg.eType := ARGTYPE_REAL;
fArg.pData := ADR(fValue);
F_BACnet_IsFinite := IsFinite(fArg);
END_FUNCTION

(* POU F_BACnet_NAN, ST *)
FUNCTION F_BACnet_NAN : REAL
(* function that generates <not-a-number> real state *)
VAR_INPUT
END_VAR
VAR
	res : POINTER TO DWORD;
END_VAR
res:=ADR(F_BACnet_NAN);
res^:=16#7FFF0000;
END_FUNCTION

(* POU F_BACnet_RealEQ, ST *)
FUNCTION F_BACnet_RealEQ : BOOL
VAR_INPUT
	fIn1	: REAL;
	fIn2	: REAL;
END_VAR
VAR
END_VAR
IF (F_BACnet_IsFinite(fIn1) <> F_BACnet_IsFinite(fIn2)) THEN
	F_BACnet_RealEQ := FALSE;
	RETURN;
END_IF
IF F_BACnet_IsFinite(fIn1) THEN
	IF (fIn1 <> fIn2) THEN
		F_BACnet_RealEQ := FALSE;
		RETURN;
	END_IF
END_IF
F_BACnet_RealEQ := TRUE;
END_FUNCTION

(* POU F_BACnet_RealGE, ST *)
FUNCTION F_BACnet_RealGE : BOOL
VAR_INPUT
	fIn1	: REAL;
	fIn2	: REAL;
END_VAR
VAR
END_VAR
IF NOT (F_BACnet_IsFinite(fIn1) OR F_BACnet_IsFinite(fIn2)) THEN
	F_BACnet_RealGE := FALSE;
	RETURN;
END_IF
F_BACnet_RealGE := (fIn1 >= fIn2);
END_FUNCTION

(* POU F_BACnet_RealGT, ST *)
FUNCTION F_BACnet_RealGT : BOOL
VAR_INPUT
	fIn1	: REAL;
	fIn2	: REAL;
END_VAR
VAR
END_VAR
IF NOT (F_BACnet_IsFinite(fIn1) OR F_BACnet_IsFinite(fIn2)) THEN
	F_BACnet_RealGT := FALSE;
	RETURN;
END_IF
F_BACnet_RealGT := (fIn1 > fIn2);
END_FUNCTION

(* POU F_BACnet_RealLE, ST *)
FUNCTION F_BACnet_RealLE : BOOL
VAR_INPUT
	fIn1	: REAL;
	fIn2	: REAL;
END_VAR
VAR
END_VAR
IF NOT (F_BACnet_IsFinite(fIn1) OR F_BACnet_IsFinite(fIn2)) THEN
	F_BACnet_RealLE := FALSE;
	RETURN;
END_IF
F_BACnet_RealLE := (fIn1 <= fIn2);
END_FUNCTION

(* POU F_BACnet_RealLT, ST *)
FUNCTION F_BACnet_RealLT : BOOL
VAR_INPUT
	fIn1	: REAL;
	fIn2	: REAL;
END_VAR
VAR
END_VAR
IF NOT (F_BACnet_IsFinite(fIn1) OR F_BACnet_IsFinite(fIn2)) THEN
	F_BACnet_RealLT := FALSE;
	RETURN;
END_IF
F_BACnet_RealLT := (fIn1 < fIn2);
END_FUNCTION

(* POU F_BACnet_RealToStr, ST *)
FUNCTION F_BACnet_RealToStr : STRING
VAR_INPUT
	pValue	: POINTER TO REAL;
END_VAR
VAR
	fArg	: T_Arg;
	pDWORD	: POINTER TO DWORD;
END_VAR
fArg.cbLen := 4;
fArg.eType := ARGTYPE_REAL;
fArg.pData := pValue;
pDWORD := pValue;
IF IsFinite(fArg) THEN
	F_BACnet_RealToStr := REAL_TO_STRING(pValue^);
ELSE
	IF (pDWORD^ AND 16#80000000) = 16#80000000 THEN
		F_BACnet_RealToStr := '-#QNAN';
	ELSE
		F_BACnet_RealToStr := '#QNAN';
	END_IF
END_IF
END_FUNCTION

(* POU F_BACnet_StatusFlags, ST *)
FUNCTION F_BACnet_StatusFlags : ST_BACnet_StatusFlags
VAR_INPUT
	data	: WORD;
END_VAR
VAR
END_VAR
F_BACnet_StatusFlags.in_alarm:= _F_BACnet_IsBitFieldBitSet( data:=data, Bit:=BACnetStatusFlags_in_alarm);
F_BACnet_StatusFlags.fault:= _F_BACnet_IsBitFieldBitSet( data:=data, Bit:=BACnetStatusFlags_fault);
F_BACnet_StatusFlags.overridden:= _F_BACnet_IsBitFieldBitSet( data:=data, Bit:=BACnetStatusFlags_overridden);
F_BACnet_StatusFlags.out_of_service:= _F_BACnet_IsBitFieldBitSet( data:=data, Bit:=BACnetStatusFlags_out_of_service);
END_FUNCTION

(* POU F_BinPV_AND, ST *)
FUNCTION F_BinPV_AND : E_BACNETBINARYPV
VAR_INPUT
	eBinPV1:	E_BACNETBINARYPV;
	eBinPV2:	E_BACNETBINARYPV;
END_VAR
VAR
END_VAR
IF (eBinPV1 = BACnetBinaryPV_NULL) AND (eBinPV2 = BACnetBinaryPV_NULL) THEN
	F_BinPV_AND := BACnetBinaryPV_NULL;
ELSIF (eBinPV1 = BACnetBinaryPV_active) AND (eBinPV2 = BACnetBinaryPV_active) THEN
	F_BinPV_AND := BACnetBinaryPV_active;
ELSE
	F_BinPV_AND := BACnetBinaryPV_inactive;
END_IF
END_FUNCTION

(* POU F_BinPV_NOT, ST *)
FUNCTION F_BinPV_NOT : E_BACNETBINARYPV
VAR_INPUT
	eBinPV:	E_BACNETBINARYPV;
END_VAR
VAR
END_VAR
IF (eBinPV = BACnetBinaryPV_NULL) THEN
	F_BinPV_NOT := BACnetBinaryPV_NULL;
ELSIF (eBinPV = BACnetBinaryPV_active) THEN
	F_BinPV_NOT := BACnetBinaryPV_inactive;
ELSE
	F_BinPV_NOT := BACnetBinaryPV_active;
END_IF
END_FUNCTION

(* POU F_BinPV_OR, ST *)
FUNCTION F_BinPV_OR : E_BACNETBINARYPV
VAR_INPUT
	eBinPV1:	E_BACNETBINARYPV;
	eBinPV2:	E_BACNETBINARYPV;
END_VAR
VAR
END_VAR
IF (eBinPV1 = BACnetBinaryPV_NULL) AND (eBinPV2 = BACnetBinaryPV_NULL) THEN
	F_BinPV_OR := BACnetBinaryPV_NULL;
ELSIF (eBinPV1 = BACnetBinaryPV_active) OR (eBinPV2 = BACnetBinaryPV_active) THEN
	F_BinPV_OR := BACnetBinaryPV_active;
ELSE
	F_BinPV_OR := BACnetBinaryPV_inactive;
END_IF
END_FUNCTION

(* POU F_BinPV_To_Bool, ST *)
FUNCTION F_BinPV_To_Bool : BOOL
VAR_INPUT
	eBinPV		: E_BACNETBINARYPV;
END_VAR
VAR
END_VAR
F_BinPV_To_Bool := (eBinPV = BACnetBinaryPV_active);
END_FUNCTION

(* POU F_BinPV_XOR, ST *)
FUNCTION F_BinPV_XOR : E_BACNETBINARYPV
VAR_INPUT
	eBinPV1:	E_BACNETBINARYPV;
	eBinPV2:	E_BACNETBINARYPV;
END_VAR
VAR
END_VAR
IF (eBinPV1 = BACnetBinaryPV_NULL) AND (eBinPV2 = BACnetBinaryPV_NULL) THEN
	F_BinPV_XOR := BACnetBinaryPV_NULL;
ELSIF (eBinPV1 = BACnetBinaryPV_active) XOR (eBinPV2 = BACnetBinaryPV_active) THEN
	F_BinPV_XOR := BACnetBinaryPV_active;
ELSE
	F_BinPV_XOR := BACnetBinaryPV_inactive;
END_IF
END_FUNCTION

(* POU F_Bool_To_BinPV, ST *)
FUNCTION F_Bool_To_BinPV : E_BACNETBINARYPV
VAR_INPUT
	bEnable	: BOOL;
	bBool	: BOOL;
END_VAR
VAR
END_VAR
IF (NOT bEnable) THEN
	F_Bool_To_BinPV := BACnetBinaryPV_NULL;
ELSIF bBOOL THEN
	F_Bool_To_BinPV := BACnetBinaryPV_active;
ELSE
	F_Bool_To_BinPV := BACnetBinaryPV_inactive;
END_IF
END_FUNCTION

(* POU F_GetVersionTcBACnet, ST *)
FUNCTION F_GetVersionTcBACnet : UINT		(* Gets the library version info *)
VAR_INPUT
	nVersionElement		: INT;
END_VAR


(* Possible nVersionElement number:
	1	:	major number
	2	:	minor number
	3	: 	revision number
*)

(* Version history:
Date		|	Version/Author			|	Created with				|	Remark
-----------------------------------------------------------------------------------------------------------------------------------
13/03/12	|	1.0.0	/ MAr			|	V2.11.0 (Build 2218)		|	* Renamed BACnet-datatype ENUM entries
20/03/12	|	1.1.0	/ MAr			|	V2.11.0 (Build 2219)		|	* Added new function blocks with ADS property write support (for WOC on local objects present_value)
			|							|								|	* Added optional input to FB_BACnet_Device to setup the valid ADS port (default 1000)
20/03/12	|	1.1.1	/ MAr			|	V2.11.0 (Build 2219)		|	* Removed obsolete flags in FB_BACnet_Program function block
27/03/12	|	1.1.2	/ MAr			|	V2.11.0 (Build 2219)		|	* FB_BACnet_ReadProp returns real processed data len (nProcessedLen)
			|							|								|	* new helper function "F_BACnet_GetObjId" added
28/03/12	|	1.1.3	/ MAr			|	V2.11.0 (Build 2219)		|	* fixed error reset in "FB_BACnet_Device"
			|							|								|	* filter object instance number in "F_BACnet_GetObjId" to prevent overflow
			|							|								|	* added ending element of BACnetObjectType-Enumeration
			|							|								|	* renamed "bErrorId" to "nErrorId" in "FB_BACnet_NotificationSinkDelEntry"
10/04/12	|	1.1.4	/ MAr			|	V2.11.0 (Build 2220)		|	* FB_BACnet_ReadProp extended with automatic handling for range properties (READ_RANGE)
21/05/12	|	1.2.0	/ MAr			|	V2.11.0 (Build 2222)		|	* Changed ENUM names to capital letter (upper case)
			|							|								|	* Renamed LOOP object process data "_SystemStatus" to "_PresentValueI"
			|							|								|	* Append update logic for remote device into remote object FBs (no need to call remote device FB explicit)
29/05/12	|	1.2.1	/ MAr			|	V2.11.0 (Build 2223)		|	* Append local object for Accumulator access (and also _EX version)
20/07/12	|	1.2.2	/ MAr			|	V2.11.0 (Build 2224)		|	* New kind of BACnet FBs "_RAW" for read/write raw values in PLC program instead of direct hardware link
			|							|								|	* Added "AckedTransitions" flags to "_EX" function blocks
			|							|								|	* Added automatic client reset to FB_BACnet_RemoteDevice (timeouts will counted, but didn't interrupt client functionality if auto-reset is active)
			|							|								|	* New time out counter as output status to FB_BACnet_RemoteDevice added
23/07/12	|	1.2.3	/ MAr			|	V2.11.0 (Build 2226)		|	* Added service fail counter to FB_BACnet_RemoteDevice
*)
CASE nVersionElement OF
	1:	F_GetVersionTcBACnet := 1;
	2:	F_GetVersionTcBACnet := 2;
	3:	F_GetVersionTcBACnet := 3;
	ELSE
		F_GetVersionTcBACnet := 16#FFFF;
END_CASE
END_FUNCTION

(* POU FB_BACnet_Accumulator, ST *)
FUNCTION_BLOCK FB_BACnet_Accumulator
VAR_INPUT
	nPV					: UDINT; (* number for present_value *)
END_VAR
VAR_IN_OUT
	Device				: FB_BACnet_Device;
END_VAR
VAR_OUTPUT
	bReady				: BOOL;
	nPresentValue		: UDINT;
	bOverridden			: BOOL;
	bOutOfService		: BOOL;
	bFault				: BOOL;
	bInAlarm			: BOOL;
	bError				: BOOL;
	nErrorId			: UINT;
END_VAR
VAR CONSTANT
	nERR_NO_ERROR		: UINT := 0;
	nERR_WRONG_MAPPING	: UINT := 2;
	nERR_OPERATIONAL	: UINT := 3;
END_VAR
VAR
	_PresentValueIn AT%I*:UDINT;	(* ~(BACnet_PresentValue	:		: )
										(BACnet_MaxPresValue	:		: writeprotect,nolink)
										(BACnet_ObjectType		: ACC	: )	*)
    _PresentValueOut AT%Q*:UDINT;	(* ~(BACnet_PresentValue	:		: )	*)
	_StatusFlags AT%I*:WORD;		(* ~(BACnet_StatusFlags		:		: )	*)
	_StatusFlagsBits : ST_BACnet_StatusFlags;

	_nUpdateCount : UDINT := 0;
END_VAR
(* update client device *)
IF Device._nUpdateCount = _nUpdateCount THEN
	Device();
END_IF
(* remind current number of update counter *)
_nUpdateCount := Device._nUpdateCount;

IF _StatusFlags < 4 THEN
	(* mapping seems to be wrong (bit string for status flags must be 4 in minimum) *)
	nErrorId := nERR_WRONG_MAPPING;

ELSIF Device.bOperational THEN
	(* clear error flag *)
	nErrorId := nERR_NO_ERROR;
	bReady := TRUE;
	(* copy present value *)
	nPresentValue 		:= _PresentValueIn;
	_PresentValueOut	:= nPV;

	(* build bit states *)
	_StatusFlagsBits	:= F_BACnet_StatusFlags(_StatusFlags);

	(* copy states to output *)
	bOverridden := _StatusFlagsBits.overridden;
	bOutOfService := _StatusFlagsBits.out_of_service;
	bFault := _StatusFlagsBits.fault;
	bInAlarm := _StatusFlagsBits.in_alarm;
ELSE
	bReady := FALSE;
	(* and set error ID *)
	nErrorId := nERR_OPERATIONAL;
END_IF

(* set error flag *)
bError := (nErrorId <> nERR_NO_ERROR);
END_FUNCTION_BLOCK

(* POU FB_BACnet_Device, ST *)
FUNCTION_BLOCK FB_BACnet_Device
VAR_INPUT
	bReset				: BOOL;
	bSupportBackup		: BOOL;
	nAdsPort			: UINT := 1000; (* Optional setting: Ads port of local BACnet-Server, default = 1000 *)
END_VAR
VAR_OUTPUT
	eSystemStatus		: E_BACNETDEVICESTATUS;
	sAmsNetId			: T_AmsNetId;
	bBackupActive		: BOOL;
	bOperational		: BOOL;
	bFirstCycle			: BOOL;
	bError				: BOOL;
	nErrorId			: UINT;
END_VAR
VAR
	_ServerControl		AT%Q*: WORD;	(* ~(BACnet_ServerControl	:		: )	*)
	_SystemStatus		AT%I*: WORD;	(* ~(BACnet_SystemStatus	:		: )
								   			(BACnet_ObjectType		: DEV	: )	*)
	_ObjIdentifier		AT%I* : DWORD;	(* ~(BACnet_ObjectIdentifier:		: LINK ) *)
	_fbWritePersistent	: FB_WritePersistentData;
	_rtrigBackup		: R_TRIG;
	_rtrigReset			: R_TRIG;

	_nPlcPort			: UINT;
	_bHasStarted		: BOOL := TRUE;

	_nUpdateCount	 	: UDINT := 0;
	_nUpdateCountAdp 	: UDINT := 0;
	_BACnetAdapter		: POINTER TO FB_BACnet_Adapter;
END_VAR
VAR CONSTANT
	nERR_NO_ERROR		: UINT := 0;
	nERR_NO_VALID_NET_ID: UINT := 1;
(* errors with reset 20.. *)
	nERR_PERSISTENT_WRITE: UINT := 20;
END_VAR
(* check pointer to bacnet adapter instance *)
IF pBACnet_Adapter > 0 THEN
	_BACnetAdapter := pBACnet_Adapter;
ELSE
	_BACnetAdapter := ADR(fbBACnet_Adapter);
END_IF

(* update adapter *)
IF _BACnetAdapter^._nUpdateCount = _nUpdateCountAdp THEN
	_BACnetAdapter^();
END_IF
(* remind current number of update counter *)
_nUpdateCountAdp := _BACnetAdapter^._nUpdateCount;

(* convert SystemStatus to enumeration *)
eSystemStatus := _SystemStatus;

(* reset trigger *)
_rtrigReset(CLK:= bReset, Q=> );
(* reset error ID and flag *)
IF (nErrorId < 20) OR _rtrigReset.Q THEN
	bError := FALSE;
	nErrorId := nERR_NO_ERROR;
END_IF

(* read NetId and convert to string *)
sAmsNetId := _BACnetAdapter^.sAmsNetId;
(* check if it plausible *)
IF sAmsNetId = '' THEN
	(* NetId not OK, return with error *)
	bError := TRUE;
	nErrorId := nERR_NO_VALID_NET_ID;
END_IF

IF ((bSupportBackup) OR _fbWritePersistent.START) THEN
	(* PLC can be backup't *)
	_ServerControl.0 := TRUE;
ELSE
	(* don't support PLC backup *)
	_ServerControl.0 := FALSE;
	_ServerControl.1 := FALSE;
END_IF

(* trigger backup flag *)
_rtrigBackup(CLK:= (eSystemStatus = BACnetDeviceStatus_BackupInProgress), Q=> );
IF _rtrigBackup.Q AND _ServerControl.0 THEN
	(* trigger backup function *)
	_fbWritePersistent.START := TRUE;
ELSIF _fbWritePersistent.START AND (NOT _fbWritePersistent.BUSY) THEN
	IF _fbWritePersistent.ERR THEN
		(* backup aborted *)
		nErrorId := nERR_PERSISTENT_WRITE;
		bError := TRUE;
	ELSE
		(* backup was successful *)
		_ServerControl.1 := TRUE;
	END_IF
ELSIF (eSystemStatus <> BACnetDeviceStatus_BackupInProgress) THEN
	(* backup process finished *)
	_ServerControl.1 := FALSE;
END_IF

(* calculate PLC runtime port *)
_nPlcPort	:= ((SystemInfo.runTimeNo - 1) * 10) + SystemInfo.runTimeNo + 800;

(* call persistent backup *)
_fbWritePersistent(
	NETID	:= '',
	PORT	:= _nPlcPort,
	START	:= ,
	TMOUT	:= ,
	MODE	:= ,
	BUSY	=> ,
	ERR		=> ,
	ERRID	=>
);

(* state *)
bBackupActive := (eSystemStatus = BACnetDeviceStatus_BackupInProgress);
bOperational :=		((eSystemStatus = BACnetDeviceStatus_Operational) AND (_BACnetAdapter^.eAdapterStatus = BACnetAdapterStatus_Complete))
				OR	(		(_BACnetAdapter^.eAdapterStatus >= BACnetAdapterStatus_GetGatewayMAC)
						AND	(_BACnetAdapter^.eAdapterStatus < BACnetAdapterStatus_Complete)
						AND	(eSystemStatus = BACnetDeviceStatus_NonOperational)
					);

(* update counter *)
IF (_nUpdateCount = 0) AND _bHasStarted THEN
	bFirstCycle := TRUE;
	_bHasStarted := FALSE;
ELSE
	bFirstCycle := FALSE;
END_IF
_nUpdateCount := _nUpdateCount +1;
END_FUNCTION_BLOCK

(* POU FB_BACnet_Adapter, ST *)
FUNCTION_BLOCK FB_BACnet_Adapter
VAR_INPUT
END_VAR
VAR_OUTPUT
	eAdapterStatus		: E_BACNETADAPTERSTATUS;
	bEthLinkOk			: BOOL;
	bGatewayOk			: BOOL;
	sAmsNetId			: T_AmsNetId;
	bFirstCycle			: BOOL;
	bError				: BOOL;
	nErrorId			: UINT;
END_VAR
VAR

	_DeviceStatus	AT%I*: WORD; (* ~(BACnet_DeviceStatus : : ) *)
	_AmsNetId		AT%I*: ARRAY[0..5] OF BYTE; (* ~(BACnet_AmsNetId : : ) *)

	_bHasStarted		: BOOL := TRUE;

	_nUpdateCount	 	: UDINT := 0;
END_VAR
VAR CONSTANT
	nERR_NO_ERROR		: UINT := 0;
	nERR_NO_VALID_NET_ID: UINT := 1;
END_VAR
(* reset error ID *)
nErrorId := nERR_NO_ERROR;

(* update bacnet adapter pointer *)
pBACnet_Adapter := ADRINST();

(* convert _DeviceStatus to enumeration *)
eAdapterStatus := SHR((_DeviceStatus AND 16#FF00), 8);

(* update netid *)
UpdateNetID();

(* states *)
bEthLinkOk := (NOT _DeviceStatus.0);
bGatewayOk := (eAdapterStatus = BACnetAdapterStatus_Complete) AND bEthLinkOk;

(* update counter *)
IF (_nUpdateCount = 0) AND _bHasStarted THEN
	bFirstCycle := TRUE;
	_bHasStarted := FALSE;
ELSE
	bFirstCycle := FALSE;
END_IF
_nUpdateCount := _nUpdateCount +1;
END_FUNCTION_BLOCK
ACTION UpdateNetID:
(* read NetId and convert to string *)
sAmsNetId := F_CreateAmsNetId(_AmsNetId);
(* check if it plausible *)
IF sAmsNetId = '0.0.0.0.0.0' THEN
	(* NetId not OK, return with error *)
	bError := TRUE;
	nErrorId := nERR_NO_VALID_NET_ID;
	sAmsNetId := '';
END_IF
END_ACTION

(* POU FB_BACnet_Accumulator_EX, ST *)
FUNCTION_BLOCK FB_BACnet_Accumulator_EX
VAR_INPUT
	nPV					: UDINT; (* number for present_value *)
END_VAR
VAR_IN_OUT
	Device				: FB_BACnet_Device;
END_VAR
VAR_OUTPUT
	bReady				: BOOL;
	nPresentValue		: UDINT;
	nMaxPV				: UDINT;
	bOverridden			: BOOL;
	bOutOfService		: BOOL;
	bFault				: BOOL;
	bInAlarm			: BOOL;
	bOverRange			: BOOL;
	bUnderRange			: BOOL;
	bNoSensor			: BOOL;
	bOpenLoop			: BOOL;
	bShortedLoop		: BOOL;
	bOtherFault			: BOOL;
	eEventState			: E_BACNETEVENTSTATE;
	bError				: BOOL;
	nErrorId			: UINT;
END_VAR
VAR CONSTANT
	nERR_NO_ERROR		: UINT := 0;
	nERR_WRONG_MAPPING	: UINT := 2;
	nERR_OPERATIONAL	: UINT := 3;
END_VAR
VAR
	_PresentValueIn AT%I*:UDINT;	(* ~(BACnet_PresentValue	:		: )
										(BACnet_ObjectType		: ACC	: )	*)
    _PresentValueOut AT%Q*:UDINT;	(* ~(BACnet_PresentValue	:		: )	*)
	_StatusFlags AT%I*:WORD;		(* ~(BACnet_StatusFlags		:		: )	*)
	_StatusFlagsBits : ST_BACnet_StatusFlags;
	_EventState AT%I*: WORD; 		(* ~(BACnet_EventState 		:		: )	*)
	_Reliability AT%I*: WORD; 		(* ~(BACnet_Reliability 	:		: )	*)
	_MaxPresValue AT%I*:UDINT;		(* ~(BACnet_MaxPresValue	:		: writeprotect) *)
	_nUpdateCount : UDINT := 0;
END_VAR
(* update client device *)
IF Device._nUpdateCount = _nUpdateCount THEN
	Device();
END_IF
(* remind current number of update counter *)
_nUpdateCount := Device._nUpdateCount;

IF _StatusFlags < 4 THEN
	(* mapping seems to be wrong (bit string for status flags must be 4 in minimum) *)
	nErrorId := nERR_WRONG_MAPPING;

ELSIF Device.bOperational THEN
	(* clear error flag *)
	nErrorId := nERR_NO_ERROR;
	bReady := TRUE;
	(* copy present value *)
	nPresentValue 		:= _PresentValueIn;
	_PresentValueOut	:= nPV;
	nMaxPV				:= _MaxPresValue;

	(* build bit states *)
	_StatusFlagsBits	:= F_BACnet_StatusFlags(_StatusFlags);

	(* copy states to output *)
	bOverridden := _StatusFlagsBits.overridden;
	bOutOfService := _StatusFlagsBits.out_of_service;
	bFault := _StatusFlagsBits.fault;
	bInAlarm := _StatusFlagsBits.in_alarm;
	bOverRange := (_Reliability = BACnetReliability_over_range);
	bUnderRange := (_Reliability = BACnetReliability_under_range);
	bNoSensor := (_Reliability = BACnetReliability_no_sensor);
	bOpenLoop := (_Reliability = BACnetReliability_open_loop);
	bShortedLoop := (_Reliability = BACnetReliability_shorted_loop);
	bOtherFault := (_Reliability = BACnetReliability_unreliable_other);

	(* convert enumeration *)
	eEventState := _EventState;
ELSE
	bReady := FALSE;
	(* and set error ID *)
	nErrorId := nERR_OPERATIONAL;
END_IF

(* set error flag *)
bError := (nErrorId <> nERR_NO_ERROR);
END_FUNCTION_BLOCK

(* POU FB_BACnet_AnalogInput, ST *)
FUNCTION_BLOCK FB_BACnet_AnalogInput
VAR_IN_OUT
	Device	: FB_BACnet_Device;
END_VAR
VAR_OUTPUT
	bReady			: BOOL;
	fPresentValue	: REAL;
	bOverridden		: BOOL;
	bOutOfService	: BOOL;
	bFault			: BOOL;
	bInAlarm		: BOOL;
	bError			: BOOL;
	nErrorId		: UINT;
END_VAR
VAR
	_PresentValue AT%I*: REAL; 			(* ~(BACnet_PresentValue 				 :		: )
								   			(BACnet_ObjectType 					 : AI	: )	*)
	_StatusFlags AT%I*: WORD; 			(* ~(BACnet_StatusFlags 				 :		: )	*)
	_StatusFlagsBits : ST_BACnet_StatusFlags;
	_nUpdateCount : UDINT := 0;
END_VAR
VAR CONSTANT
	nERR_NO_ERROR		: UINT := 0;
	nERR_WRONG_MAPPING	: UINT := 2;
	nERR_OPERATIONAL	: UINT := 3;
END_VAR
(* update server device *)
IF Device._nUpdateCount = _nUpdateCount THEN
	Device();
END_IF
(* remind current number of update counter *)
_nUpdateCount := Device._nUpdateCount;

(* check BitString format of StatusFlags --> if StatusFlags are less than 4, object isn't linked correctly *)
IF (_StatusFlags < 4) THEN
	(* wrong mapping *)
	nErrorId := nERR_WRONG_MAPPING;
	bReady := FALSE;

ELSIF Device.bOperational THEN
	(* ready state *)
	bReady := TRUE;
	nErrorId := nERR_NO_ERROR;

	(* present value *)
	fPresentValue := _PresentValue;

	(* build bit states *)
	_StatusFlagsBits := F_BACnet_StatusFlags(_StatusFlags);

	(* copy states to output *)
	bOverridden := _StatusFlagsBits.overridden;
	bOutOfService := _StatusFlagsBits.out_of_service;
	bFault := _StatusFlagsBits.fault;
	bInAlarm := _StatusFlagsBits.in_alarm;
ELSE
	(* server device not ready, reset local ready also *)
	bReady := FALSE;
	nErrorId := nERR_OPERATIONAL;
END_IF
(* set error flag *)
bError := (nErrorId <> nERR_NO_ERROR);
END_FUNCTION_BLOCK

(* POU FB_BACnet_AnalogInput_EX, ST *)
FUNCTION_BLOCK FB_BACnet_AnalogInput_EX
VAR_IN_OUT
	Device	: FB_BACnet_Device;
END_VAR
VAR_OUTPUT
	bReady			: BOOL;
	fPresentValue	: REAL;
	bOverridden		: BOOL;
	bOutOfService	: BOOL;
	bFault			: BOOL;
	bInAlarm		: BOOL;
	bOverRange		: BOOL;
	bUnderRange		: BOOL;
	bNoSensor		: BOOL;
	bOpenLoop		: BOOL;
	bShortedLoop	: BOOL;
	bOtherFault		: BOOL;
	eEventState		: E_BACNETEVENTSTATE;
	bAckedTrans_ToOffNormal : BOOL;
	bAckedTrans_ToFault		: BOOL;
	bAckedTrans_ToNormal	: BOOL;
	bError			: BOOL;
	nErrorId		: UINT;
END_VAR
VAR
	_PresentValue AT%I*: REAL; 			(* ~(BACnet_PresentValue 				 :		: )
								   			(BACnet_ObjectType 					 : AI	: )	*)
	_StatusFlags AT%I*: WORD; 			(* ~(BACnet_StatusFlags 				 :		: )	*)
	_StatusFlagsBits : ST_BACnet_StatusFlags;
	_EventState AT%I*: WORD; 			(* ~(BACnet_EventState 					 :		: )	*)
	_Reliability AT%I*: WORD; 			(* ~(BACnet_Reliability 				 :		: )	*)
	_AckedTransitions AT%I*:WORD;		(* ~(BACnet_AckedTransitions:		: ) *)
	_AckedTransBits : ST_BACnet_EventTransitionBits;
	_nUpdateCount : UDINT := 0;
END_VAR
VAR CONSTANT
	nERR_NO_ERROR		: UINT := 0;
	nERR_WRONG_MAPPING	: UINT := 2;
	nERR_OPERATIONAL	: UINT := 3;
END_VAR
(* update server device *)
IF Device._nUpdateCount = _nUpdateCount THEN
	Device();
END_IF
(* remind current number of update counter *)
_nUpdateCount := Device._nUpdateCount;

(* check BitString format of StatusFlags --> if StatusFlags are less than 4, object isn't linked correctly *)
IF (_StatusFlags < 4) OR _AckedTransitions < 5 THEN
	(* wrong mapping *)
	nErrorId := nERR_WRONG_MAPPING;
	bReady := FALSE;

ELSIF Device.bOperational THEN
	(* ready state *)
	bReady := TRUE;
	nErrorId := nERR_NO_ERROR;

	(* present value *)
	fPresentValue := _PresentValue;

	(* build bit states *)
	_StatusFlagsBits := F_BACnet_StatusFlags(_StatusFlags);
	_AckedTransBits		:= F_BACnet_EventTransitionFlags(_AckedTransitions);

	(* copy states to output *)
	bOverridden := _StatusFlagsBits.overridden;
	bOutOfService := _StatusFlagsBits.out_of_service;
	bFault := _StatusFlagsBits.fault;
	bInAlarm := _StatusFlagsBits.in_alarm;
	bOverRange := (_Reliability = BACnetReliability_over_range);
	bUnderRange := (_Reliability = BACnetReliability_under_range);
	bNoSensor := (_Reliability = BACnetReliability_no_sensor);
	bOpenLoop := (_Reliability = BACnetReliability_open_loop);
	bShortedLoop := (_Reliability = BACnetReliability_shorted_loop);
	bOtherFault := (_Reliability = BACnetReliability_unreliable_other);
	bAckedTrans_ToOffNormal := _AckedTransBits.to_offnormal;
	bAckedTrans_ToFault := _AckedTransBits.to_fault;
	bAckedTrans_ToNormal := _AckedTransBits.to_normal;

	(* convert enumeration *)
	eEventState := _EventState;
ELSE
	(* server device not ready, reset local ready also *)
	bReady := FALSE;
	nErrorId := nERR_OPERATIONAL;
END_IF
(* set error flag *)
bError := (nErrorId <> nERR_NO_ERROR);
END_FUNCTION_BLOCK

(* POU FB_BACnet_AnalogInput_RAW, ST *)
FUNCTION_BLOCK FB_BACnet_AnalogInput_RAW
VAR_INPUT
	nRawIn			AT%Q*: INT;(* ~(BACnet_RawIoAnalogSignedValue : : ) *)
END_VAR
VAR_IN_OUT
	Device	: FB_BACnet_Device;
END_VAR
VAR_OUTPUT
	bReady			: BOOL;
	fPresentValue	: REAL;
	bOverridden		: BOOL;
	bOutOfService	: BOOL;
	bFault			: BOOL;
	bInAlarm		: BOOL;
	bAckedTrans_ToOffNormal : BOOL;
	bAckedTrans_ToFault		: BOOL;
	bAckedTrans_ToNormal	: BOOL;
	bError			: BOOL;
	nErrorId		: UINT;
END_VAR
VAR
	_PresentValue AT%I*: REAL; 			(* ~(BACnet_PresentValue 				 :		: )
								   			(BACnet_ObjectType 					 : AI	: )	*)
	_StatusFlags AT%I*: WORD; 			(* ~(BACnet_StatusFlags 				 :		: )	*)
	_AckedTransitions AT%I*:WORD;		(* ~(BACnet_AckedTransitions:		: ) *)
	_AckedTransBits : ST_BACnet_EventTransitionBits;
	_StatusFlagsBits : ST_BACnet_StatusFlags;
	_nUpdateCount : UDINT := 0;
END_VAR
VAR CONSTANT
	nERR_NO_ERROR		: UINT := 0;
	nERR_WRONG_MAPPING	: UINT := 2;
	nERR_OPERATIONAL	: UINT := 3;
END_VAR
(* update server device *)
IF Device._nUpdateCount = _nUpdateCount THEN
	Device();
END_IF
(* remind current number of update counter *)
_nUpdateCount := Device._nUpdateCount;

(* check BitString format of StatusFlags --> if StatusFlags are less than 4, object isn't linked correctly *)
IF (_StatusFlags < 4) OR _AckedTransitions < 5 THEN
	(* wrong mapping *)
	nErrorId := nERR_WRONG_MAPPING;
	bReady := FALSE;

ELSIF Device.bOperational THEN
	(* ready state *)
	bReady := TRUE;
	nErrorId := nERR_NO_ERROR;

	(* present value *)
	fPresentValue := _PresentValue;

	(* build bit states *)
	_StatusFlagsBits := F_BACnet_StatusFlags(_StatusFlags);
	_AckedTransBits		:= F_BACnet_EventTransitionFlags(_AckedTransitions);

	(* copy states to output *)
	bOverridden := _StatusFlagsBits.overridden;
	bOutOfService := _StatusFlagsBits.out_of_service;
	bFault := _StatusFlagsBits.fault;
	bInAlarm := _StatusFlagsBits.in_alarm;
	bAckedTrans_ToOffNormal := _AckedTransBits.to_offnormal;
	bAckedTrans_ToFault := _AckedTransBits.to_fault;
	bAckedTrans_ToNormal := _AckedTransBits.to_normal;
ELSE
	(* server device not ready, reset local ready also *)
	bReady := FALSE;
	nErrorId := nERR_OPERATIONAL;
END_IF
(* set error flag *)
bError := (nErrorId <> nERR_NO_ERROR);
END_FUNCTION_BLOCK

(* POU FB_BACnet_AnalogOutput, ST *)
FUNCTION_BLOCK FB_BACnet_AnalogOutput
VAR_INPUT
	bEnablePV		: BOOL; (* enable present value with priority x in priority array, FALSE = priority x disable *)
	fPV		: REAL; (* decimal number for priority x, when input bEnablePV is TRUE *)
END_VAR
VAR_IN_OUT
	Device	: FB_BACnet_Device;
END_VAR
VAR_OUTPUT
	bReady			: BOOL;
	fPresentValue	: REAL;
	bOverridden		: BOOL;
	bOutOfService	: BOOL;
	bFault			: BOOL;
	bInAlarm		: BOOL;
	bError			: BOOL;
	nErrorId		: UINT;
END_VAR
VAR
	_PresentValue AT%I*: REAL; 			(* ~(BACnet_PresentValue 				 :		: )
								   			(BACnet_ObjectType 					 : AO	: )	*)
    _PresentValue_Priority12 AT%Q*: REAL;(* ~(BACnet_PresentValue_Priority12 	 	 :		: )	*)
	_StatusFlags AT%I*: WORD; 			(* ~(BACnet_StatusFlags 				 :		: )	*)
	_StatusFlagsBits : ST_BACnet_StatusFlags;
	_nUpdateCount : UDINT := 0;
END_VAR
VAR CONSTANT
	nERR_NO_ERROR		: UINT := 0;
	nERR_WRONG_MAPPING	: UINT := 2;
	nERR_OPERATIONAL	: UINT := 3;
END_VAR
(* update server device *)
IF Device._nUpdateCount = _nUpdateCount THEN
	Device();
END_IF
(* remind current number of update counter *)
_nUpdateCount := Device._nUpdateCount;

(* check BitString format of StatusFlags --> if StatusFlags are less than 4, object isn't linked correctly *)
IF (_StatusFlags < 4) THEN
	(* wrong mapping *)
	nErrorId := nERR_WRONG_MAPPING;
	bReady := FALSE;

ELSIF Device.bOperational THEN
	(* ready state *)
	bReady := TRUE;
	nErrorId := nERR_NO_ERROR;

	(* write into priority array *)
	IF bEnablePV THEN
		_PresentValue_Priority12	:= fPV;
	ELSE
		_PresentValue_Priority12	:= F_BACnet_NAN();
	END_IF

	(* present value *)
	fPresentValue := _PresentValue;

	(* build bit states *)
	_StatusFlagsBits := F_BACnet_StatusFlags(_StatusFlags);

	(* copy states to output *)
	bOverridden := _StatusFlagsBits.overridden;
	bOutOfService := _StatusFlagsBits.out_of_service;
	bFault := _StatusFlagsBits.fault;
	bInAlarm := _StatusFlagsBits.in_alarm;

ELSIF Device.bFirstCycle THEN
	(* first call of the server device since reboot/reset *)
	bReady := FALSE;
	_PresentValue_Priority12 := F_BACnet_NAN();
ELSE
	(* server device not ready, reset local ready also *)
	bReady := FALSE;
	nErrorId := nERR_OPERATIONAL;
END_IF
(* set error flag *)
bError := (nErrorId <> nERR_NO_ERROR);
END_FUNCTION_BLOCK

(* POU FB_BACnet_AnalogOutput_ADS, ST *)
FUNCTION_BLOCK FB_BACnet_AnalogOutput_ADS
VAR_INPUT
	bEnablePV		: BOOL;
	fPV				: REAL; (* decimal number for priority x, when input bEnablePV is TRUE *)
	bManual			: BOOL; (* FALSE --> TRUE: write present_value immediately, FALSE: only write present_value on-change, TRUE: write present_value on-change and when device turns operational *)
	ePriority		: E_BACNETPRIORITY := BACNETPRIORITY_12;
END_VAR
VAR_IN_OUT
	Device			: FB_BACnet_Device;
END_VAR
VAR_OUTPUT
	bReady			: BOOL;
	bPvDone			: BOOL; (* present_value written over ADS *)
	fPresentValue	: REAL;
	bOverridden		: BOOL;
	bOutOfService	: BOOL;
	bFault			: BOOL;
	bInAlarm		: BOOL;
	bError			: BOOL;
	nErrorId		: UINT;
	nAdsErrorId		: UDINT;
END_VAR
VAR
	_PresentValue AT%I*: REAL; 			(* ~(BACnet_PresentValue 				 :		: )
								   			(BACnet_ObjectType 					 : AO	: )	*)
    _PresentValue_Ads : REAL;
	_StatusFlags AT%I*: WORD; 			(* ~(BACnet_StatusFlags 				 :		: )	*)
	_ObjectId AT%I*: DWORD;				(* ~(BACnet_ObjectIdentifier			 :		: LINK) *)
	_StatusFlagsBits : ST_BACnet_StatusFlags;
	_nUpdateCount : UDINT := 0;
	_WriteProp : FB_BACnet_WriteProp;
	_rtrigManual : R_TRIG;
	_bEnPvOld : BOOL;
	_nObjType : E_BACNETOBJECTTYPE;
END_VAR
VAR CONSTANT
	nERR_NO_ERROR		: UINT := 0;
	nERR_WRONG_MAPPING	: UINT := 2;
	nERR_OPERATIONAL	: UINT := 3;
	nERR_WRONG_TYPE		: UINT := 4;
END_VAR
(* update server device *)
IF Device._nUpdateCount = _nUpdateCount THEN
	Device();
END_IF
(* remind current number of update counter *)
_nUpdateCount := Device._nUpdateCount;

(* trigger on manual flag *)
_rtrigManual(CLK:= bManual, Q=> );

(* decode object type *)
_nObjType := F_BACnet_GetObjType(_ObjectId);

(* check BitString format of StatusFlags --> if StatusFlags are less than 4, object isn't linked correctly *)
IF _nObjType <> BACnetObjectType_AnalogOutput THEN
	(* wrong mapped object type *)
	nErrorId := nERR_WRONG_TYPE;
	bReady := FALSE;
	bPvDone := FALSE;

ELSIF (_StatusFlags < 4) THEN
	(* wrong mapping *)
	nErrorId := nERR_WRONG_MAPPING;
	bReady := FALSE;
	bPvDone := FALSE;

ELSIF Device.bOperational THEN
	(* write present_value on manual trigger, on-change and on operational recover *)
	IF		_rtrigManual.Q
		OR	((NOT F_BACnet_RealEQ(fPV, _PresentValue_Ads)) AND bEnablePV)
		OR	((NOT bReady) AND bManual)
		OR	(bEnablePV <> _bEnPvOld)
	THEN
		_WriteProp.bExecute := TRUE;
		bPvDone := FALSE;
		(* write depending on enable state *)
		IF bEnablePV THEN
			_PresentValue_Ads := fPV;
		ELSE
			_PresentValue_Ads := F_BACnet_NAN();
		END_IF
		_bEnPvOld := bEnablePV;
	END_IF

	(* ready state *)
	bReady := TRUE;
	nErrorId := nERR_NO_ERROR;

	(* present value *)
	fPresentValue := _PresentValue;

	(* build bit states *)
	_StatusFlagsBits := F_BACnet_StatusFlags(_StatusFlags);

	(* copy states to output *)
	bOverridden := _StatusFlagsBits.overridden;
	bOutOfService := _StatusFlagsBits.out_of_service;
	bFault := _StatusFlagsBits.fault;
	bInAlarm := _StatusFlagsBits.in_alarm;

ELSIF Device.bFirstCycle THEN
	(* first call of the server device since reboot/reset *)
	bReady := FALSE;
	bPvDone := FALSE;
ELSE
	(* server device not ready, reset local ready also *)
	bReady := FALSE;
	nErrorId := nERR_OPERATIONAL;
	bPvDone := FALSE;
END_IF

(* call write property command *)
_WriteProp(
	BACnetDevicePort	:= Device.nAdsPort,
	bExecute			:= ,
	sNetId				:= Device.sAmsNetId,
	ObjectType			:= _nObjType,
	PropertyID			:= BACnetPropertyIdentifier_PresentValue,
	Priority			:= ePriority,
	DataType			:= BACnetDataType_Real,
	ObjectInstance		:= F_BACnet_GetObjInstance(_ObjectId),
	ptrValue			:= ADR(_PresentValue_Ads),
	nLenValue			:= SIZEOF(_PresentValue_Ads),
	bDone				=> ,
	bBusy				=> ,
	bError				=> ,
	nErrID				=> nAdsErrorId);

(* set done flag *)
IF _WriteProp.bExecute AND (NOT _WriteProp.bBusy) THEN
	(* reset execution bit *)
	_WriteProp(bExecute := FALSE);
	(* check if command was finished with error *)
	IF _WriteProp.bError THEN
		IF bManual THEN
			(* retrigger if manual flag is set *)
			_WriteProp.bExecute := TRUE;
		END_IF
		bPvDone := FALSE;
	ELSE
		(* successful written *)
		bPvDone	:= TRUE;
	END_IF
END_IF

(* set error flag *)
bError := (nErrorId <> nERR_NO_ERROR) OR (nAdsErrorId <> 0);
END_FUNCTION_BLOCK

(* POU FB_BACnet_WriteProp, ST *)
FUNCTION_BLOCK FB_BACnet_WriteProp
VAR_INPUT
	BACnetDevicePort	: UINT := 16#FFFF;
	bExecute			: BOOL;
	sNetId				: T_AmsNetId;
	ObjectType			: E_BACNETOBJECTTYPE;
	PropertyID			: E_BACNETPROPERTYIDENTIFIER;
	Priority			: E_BACNETPRIORITY;
	DataType			: E_BACNETDATATYPES;
	ObjectInstance		: UDINT;
	ptrValue			: POINTER TO BYTE;
	nLenValue			: UDINT; (* byte size of value (SIZEOF) *)
END_VAR
VAR_OUTPUT
	bDone				: BOOL;
	bBusy				: BOOL;
	bError				: BOOL;
	nErrID				: UDINT;
END_VAR
VAR
	_Write				: ADSWRITE;
	_rtrigStart			: R_TRIG;
	_len_data			: UDINT;
	_nPrio 				: UDINT;
	_ptrDWORD			: POINTER TO DWORD;
	_ptrREAL			: POINTER TO REAL;
	_ptrBYTE			: POINTER TO BYTE;
	_dataPointer		: POINTER TO BYTE;
	_dwordVal			: DWORD;
END_VAR
(* catch the start flag *)
	_rtrigStart(Clk:=bExecute);

(* prepare *)
	IF _rtrigStart.Q AND (NOT bBusy) THEN
		_Write(WRITE := FALSE);
		bDone := FALSE;
		bBusy := TRUE;
		bError := FALSE;
		nErrId := 0;
		_nPrio := SHL(INT_TO_UDINT(Priority), 26);
		_len_data := nLenValue; (* in default, take the user given length *)
		_dataPointer := ptrValue;
		CASE DataType OF
			BACnetDataType_Null 				: _len_data := 0; (* set length to zero *)
			BACnetDataType_Bool 				: _len_data := _len_data; (* 1 *)
			BACnetDataType_CharacterStringExt	: _len_data := _len_data; (* 2 *)

			BACnetDataType_UnsignedInteger,
			BACnetDataType_SignedInteger 		: _len_data := MIN(_len_data, 4); (* 4 *)
				IF (_len_data >= 4) THEN
					(* source data type bigger/equal 4 byte --> OK, take first 4 byte *)
					_ptrDWORD := ptrValue;
				ELSE
					(* upgrade data type from less 4 byte to fully double word *)
					_dwordVal := 0;
					_ptrDWORD := ADR(_dwordVal);
					MEMCPY(destAddr:=_ptrDWORD, srcAddr:=ptrValue, n:=_len_data);
					_dataPointer := _ptrDWORD; (* from here on, point to the internal data source *)
					_len_data := SIZEOF(_dwordVal); (* increase size to internal data type length *)
				END_IF
				(* make some plausibility checks *)
				IF	(		ObjectType = BACnetObjectType_MultiStateInput
						OR	ObjectType = BACnetObjectType_MultiStateOutput
						OR	ObjectType = BACnetObjectType_MultiStateValue
					)
				THEN
					IF _ptrDWORD^ = 0 THEN
						(* set data type and data length to NULL operation *)
						_len_data := 0;
					END_IF
				END_IF

			BACnetDataType_Real 				: _len_data := _len_data; (* 4 *)
				_ptrREAL := ptrValue;
				IF (NOT F_BACnet_IsFinite(_ptrREAL^)) THEN
					(* set data type and data length to NULL operation *)
					_len_data := 0;
				END_IF

			BACnetDataType_Double 				: _len_data := _len_data; (* 8 *)
			BACnetDataType_OctetString 			: _len_data := _len_data; (* 8 *)
			BACnetDataType_Enumerated 			: _len_data := _len_data; (* 8 *)
			BACnetDataType_LimitEnable			: _len_data := _len_data; (* 4 *)
			BACnetDataType_BitString 			: _len_data := _len_data; (* 11 *)

			BACnetDataType_BinaryPV				: _len_data := MIN(_len_data, 1); (* 1 *)
				_ptrByte := ptrValue;
				IF		_len_data <= 0
					OR	_ptrByte^ >= 2
				THEN
					_len_data := 0;
				END_IF

		END_CASE;
	END_IF;

(* execute *)
	IF bBusy THEN
		_Write(	NETID:= sNetId,
				PORT:= BACnetDevicePort,
				IDXGRP:=16#80000000 + INT_TO_UDINT(PropertyID) + _nPrio,
				IDXOFFS:= ObjectInstance + SHL(INT_TO_UDINT(ObjectType), 22),
				LEN:= _len_data,
				SRCADDR:= _dataPointer,
				WRITE:= TRUE,
				TMOUT:= tBACnet_ADSTimeOut);
		IF NOT _Write.Busy THEN
			IF _Write.Err THEN
				nErrID := _Write.ErrId;
				bError := TRUE;
			END_IF
			_Write(WRITE := FALSE);
			bBusy := FALSE;
			bDone := NOT bError;
		END_IF
	END_IF
END_FUNCTION_BLOCK

(* POU FB_BACnet_AnalogOutput_EX, ST *)
FUNCTION_BLOCK FB_BACnet_AnalogOutput_EX
VAR_INPUT
	bEnablePV		: BOOL; (* enable present value with priority x in priority array, FALSE = priority x disable *)
	fPV		: REAL; (* decimal number for priority x, when input bEnablePV is TRUE *)
END_VAR
VAR_IN_OUT
	Device	: FB_BACnet_Device;
END_VAR
VAR_OUTPUT
	bReady			: BOOL;
	fPresentValue	: REAL;
	bOverridden		: BOOL;
	bOutOfService	: BOOL;
	bFault			: BOOL;
	bInAlarm		: BOOL;
	bNoOutput		: BOOL;
	bOpenLoop		: BOOL;
	bShortedLoop	: BOOL;
	bOtherFault		: BOOL;
	eEventState		: E_BACNETEVENTSTATE;
	bAckedTrans_ToOffNormal : BOOL;
	bAckedTrans_ToFault		: BOOL;
	bAckedTrans_ToNormal	: BOOL;
	nActivePrio		: UINT;
	bError			: BOOL;
	nErrorId		: UINT;
END_VAR
VAR
	_PresentValue AT%I*: REAL; 			(* ~(BACnet_PresentValue 				 :		: )
								   			(BACnet_ObjectType 					 : AO	: )	*)
    _PresentValue_Priority12 AT%Q*: REAL;(* ~(BACnet_PresentValue_Priority12 	 	 :		: )	*)
	_StatusFlags AT%I*: WORD; 			(* ~(BACnet_StatusFlags 				 :		: )	*)
	_StatusFlagsBits : ST_BACnet_StatusFlags;
	_EventState AT%I*: WORD;			(* ~(BACnet_EventState 					 :		: )	*)
	_Reliability AT%I*: WORD; 			(* ~(BACnet_Reliability 				 :		: )	*)
	_ActivePriority AT%I*: UDINT; 		(* ~(BACnet_ActivePriority 				 :		: )	*)
	_AckedTransitions AT%I*:WORD;		(* ~(BACnet_AckedTransitions:		: ) *)
	_AckedTransBits : ST_BACnet_EventTransitionBits;
	_nUpdateCount : UDINT := 0;
END_VAR
VAR CONSTANT
	nERR_NO_ERROR		: UINT := 0;
	nERR_WRONG_MAPPING	: UINT := 2;
	nERR_OPERATIONAL	: UINT := 3;
END_VAR
(* update server device *)
IF Device._nUpdateCount = _nUpdateCount THEN
	Device();
END_IF
(* remind current number of update counter *)
_nUpdateCount := Device._nUpdateCount;

(* check BitString format of StatusFlags --> if StatusFlags are less than 4, object isn't linked correctly *)
IF (_StatusFlags < 4) OR _AckedTransitions < 5 THEN
	(* wrong mapping *)
	nErrorId := nERR_WRONG_MAPPING;
	bReady := FALSE;

ELSIF Device.bOperational THEN
	(* ready state *)
	bReady := TRUE;
	nErrorId := nERR_NO_ERROR;

	(* write into priority array *)
	IF bEnablePV THEN
		_PresentValue_Priority12	:= fPV;
	ELSE
		_PresentValue_Priority12	:= F_BACnet_NAN();
	END_IF

	(* present value *)
	fPresentValue := _PresentValue;

	(* build bit states *)
	_StatusFlagsBits := F_BACnet_StatusFlags(_StatusFlags);
	_AckedTransBits		:= F_BACnet_EventTransitionFlags(_AckedTransitions);

	(* copy states to output *)
	bOverridden := _StatusFlagsBits.overridden;
	bOutOfService := _StatusFlagsBits.out_of_service;
	bFault := _StatusFlagsBits.fault;
	bInAlarm := _StatusFlagsBits.in_alarm;
	bNoOutput := (_Reliability = BACnetReliability_no_output);
	bOpenLoop := (_Reliability = BACnetReliability_open_loop);
	bShortedLoop := (_Reliability = BACnetReliability_shorted_loop);
	bOtherFault := (_Reliability = BACnetReliability_unreliable_other);
	bAckedTrans_ToOffNormal := _AckedTransBits.to_offnormal;
	bAckedTrans_ToFault := _AckedTransBits.to_fault;
	bAckedTrans_ToNormal := _AckedTransBits.to_normal;

	(* convert enumeration *)
	eEventState := _EventState;

	(* copy active priority *)
	nActivePrio := UDINT_TO_UINT(_ActivePriority);

ELSIF Device.bFirstCycle THEN
	(* first call of the server device since reboot/reset *)
	bReady := FALSE;
	_PresentValue_Priority12 := F_BACnet_NAN();
ELSE
	(* server device not ready, reset local ready also *)
	bReady := FALSE;
	nErrorId := nERR_OPERATIONAL;
END_IF
(* set error flag *)
bError := (nErrorId <> nERR_NO_ERROR);
END_FUNCTION_BLOCK

(* POU FB_BACnet_AnalogOutput_RAW, ST *)
FUNCTION_BLOCK FB_BACnet_AnalogOutput_RAW
VAR_INPUT
	bEnablePV		: BOOL; (* enable present value with priority x in priority array, FALSE = priority x disable *)
	fPV		: REAL; (* decimal number for priority x, when input bEnablePV is TRUE *)
END_VAR
VAR_IN_OUT
	Device	: FB_BACnet_Device;
END_VAR
VAR_OUTPUT
	bReady			: BOOL;
	fPresentValue	: REAL;
	bOverridden		: BOOL;
	bOutOfService	: BOOL;
	bFault			: BOOL;
	bInAlarm		: BOOL;
	bAckedTrans_ToOffNormal : BOOL;
	bAckedTrans_ToFault		: BOOL;
	bAckedTrans_ToNormal	: BOOL;
	bError			: BOOL;
	nErrorId		: UINT;
	nRawOut			AT%I*: INT;(* ~(BACnet_RawIoAnalogSignedValue : : ) *)
END_VAR
VAR
	_PresentValue AT%I*: REAL; 			(* ~(BACnet_PresentValue 				 :		: )
								   			(BACnet_ObjectType 					 : AO	: )	*)
    _PresentValue_Priority12 AT%Q*: REAL;(* ~(BACnet_PresentValue_Priority12 	 	 :		: )	*)
	_StatusFlags AT%I*: WORD; 			(* ~(BACnet_StatusFlags 				 :		: )	*)
	_AckedTransitions AT%I*:WORD;		(* ~(BACnet_AckedTransitions:		: ) *)
	_AckedTransBits : ST_BACnet_EventTransitionBits;
	_StatusFlagsBits : ST_BACnet_StatusFlags;
	_nUpdateCount : UDINT := 0;
END_VAR
VAR CONSTANT
	nERR_NO_ERROR		: UINT := 0;
	nERR_WRONG_MAPPING	: UINT := 2;
	nERR_OPERATIONAL	: UINT := 3;
END_VAR
(* update server device *)
IF Device._nUpdateCount = _nUpdateCount THEN
	Device();
END_IF
(* remind current number of update counter *)
_nUpdateCount := Device._nUpdateCount;

(* check BitString format of StatusFlags --> if StatusFlags are less than 4, object isn't linked correctly *)
IF (_StatusFlags < 4) OR _AckedTransitions < 5 THEN
	(* wrong mapping *)
	nErrorId := nERR_WRONG_MAPPING;
	bReady := FALSE;

ELSIF Device.bOperational THEN
	(* ready state *)
	bReady := TRUE;
	nErrorId := nERR_NO_ERROR;

	(* write into priority array *)
	IF bEnablePV THEN
		_PresentValue_Priority12	:= fPV;
	ELSE
		_PresentValue_Priority12	:= F_BACnet_NAN();
	END_IF

	(* present value *)
	fPresentValue := _PresentValue;

	(* build bit states *)
	_StatusFlagsBits := F_BACnet_StatusFlags(_StatusFlags);
	_AckedTransBits		:= F_BACnet_EventTransitionFlags(_AckedTransitions);

	(* copy states to output *)
	bOverridden := _StatusFlagsBits.overridden;
	bOutOfService := _StatusFlagsBits.out_of_service;
	bFault := _StatusFlagsBits.fault;
	bInAlarm := _StatusFlagsBits.in_alarm;
	bAckedTrans_ToOffNormal := _AckedTransBits.to_offnormal;
	bAckedTrans_ToFault := _AckedTransBits.to_fault;
	bAckedTrans_ToNormal := _AckedTransBits.to_normal;

ELSIF Device.bFirstCycle THEN
	(* first call of the server device since reboot/reset *)
	bReady := FALSE;
	_PresentValue_Priority12 := F_BACnet_NAN();
ELSE
	(* server device not ready, reset local ready also *)
	bReady := FALSE;
	nErrorId := nERR_OPERATIONAL;
END_IF
(* set error flag *)
bError := (nErrorId <> nERR_NO_ERROR);
END_FUNCTION_BLOCK

(* POU FB_BACnet_AnalogValue, ST *)
FUNCTION_BLOCK FB_BACnet_AnalogValue
VAR_INPUT
	bEnablePV		: BOOL; (* enable present value with priority x in priority array, FALSE = priority x disable *)
	fPV		: REAL; (* decimal number for priority x, when input bEnablePV is TRUE *)
END_VAR
VAR_IN_OUT
	Device	: FB_BACnet_Device;
END_VAR
VAR_OUTPUT
	bReady			: BOOL;
	fPresentValue	: REAL;
	bOverridden		: BOOL;
	bOutOfService	: BOOL;
	bFault			: BOOL;
	bInAlarm		: BOOL;
	bError			: BOOL;
	nErrorId		: UINT;
END_VAR
VAR
	_PresentValue AT%I*: REAL; 			(* ~(BACnet_PresentValue 				:		: )
								   			(BACnet_ObjectType 					: AV	: )	*)
    _PresentValue_Priority12 AT%Q*: REAL;(* ~(BACnet_PresentValue_Priority12		:		: )	*)
	_StatusFlags AT%I*: WORD; 			(* ~(BACnet_StatusFlags 				:		: )	*)
	_StatusFlagsBits : ST_BACnet_StatusFlags;
	_nUpdateCount : UDINT := 0;
END_VAR
VAR CONSTANT
	nERR_NO_ERROR		: UINT := 0;
	nERR_WRONG_MAPPING	: UINT := 2;
	nERR_OPERATIONAL	: UINT := 3;
END_VAR
(* update server device *)
IF Device._nUpdateCount = _nUpdateCount THEN
	Device();
END_IF
(* remind current number of update counter *)
_nUpdateCount := Device._nUpdateCount;

(* check BitString format of StatusFlags --> if StatusFlags are less than 4, object isn't linked correctly *)
IF (_StatusFlags < 4) THEN
	(* wrong mapping *)
	nErrorId := nERR_WRONG_MAPPING;
	bReady := FALSE;

ELSIF Device.bOperational THEN
	(* ready state *)
	bReady := TRUE;
	nErrorId := nERR_NO_ERROR;

	(* write into priority array *)
	IF bEnablePV THEN
		_PresentValue_Priority12	:= fPV;
	ELSE
		_PresentValue_Priority12	:= F_BACnet_NAN();
	END_IF

	(* present value *)
	fPresentValue := _PresentValue;

	(* build bit states *)
	_StatusFlagsBits := F_BACnet_StatusFlags(_StatusFlags);

	(* copy states to output *)
	bOverridden := _StatusFlagsBits.overridden;
	bOutOfService := _StatusFlagsBits.out_of_service;
	bFault := _StatusFlagsBits.fault;
	bInAlarm := _StatusFlagsBits.in_alarm;

ELSIF Device.bFirstCycle THEN
	(* first call of the server device since reboot/reset *)
	bReady := FALSE;
	_PresentValue_Priority12 := F_BACnet_NAN();
ELSE
	(* server device not ready, reset local ready also *)
	bReady := FALSE;
	nErrorId := nERR_OPERATIONAL;
END_IF
(* set error flag *)
bError := (nErrorId <> nERR_NO_ERROR);
END_FUNCTION_BLOCK

(* POU FB_BACnet_AnalogValue_ADS, ST *)
FUNCTION_BLOCK FB_BACnet_AnalogValue_ADS
VAR_INPUT
	bEnablePV		: BOOL;
	fPV				: REAL; (* decimal number for priority x, when input bEnablePV is TRUE *)
	bManual			: BOOL; (* FALSE --> TRUE: write present_value immediately, FALSE: only write present_value on-change, TRUE: write present_value on-change and when device turns operational *)
	ePriority		: E_BACNETPRIORITY := BACNETPRIORITY_12;
END_VAR
VAR_IN_OUT
	Device			: FB_BACnet_Device;
END_VAR
VAR_OUTPUT
	bReady			: BOOL;
	bPvDone			: BOOL; (* present_value written over ADS *)
	fPresentValue	: REAL;
	bOverridden		: BOOL;
	bOutOfService	: BOOL;
	bFault			: BOOL;
	bInAlarm		: BOOL;
	bError			: BOOL;
	nErrorId		: UINT;
	nAdsErrorId		: UDINT;
END_VAR
VAR
	_PresentValue AT%I*: REAL; 			(* ~(BACnet_PresentValue 				:		: )
								   			(BACnet_ObjectType 					: AV	: )	*)
    _PresentValue_Ads : REAL;
	_StatusFlags AT%I*: WORD; 			(* ~(BACnet_StatusFlags 				:		: )	*)
	_ObjectId AT%I*: DWORD;				(* ~(BACnet_ObjectIdentifier			 :		: LINK) *)
	_StatusFlagsBits : ST_BACnet_StatusFlags;
	_nUpdateCount : UDINT := 0;
	_WriteProp : FB_BACnet_WriteProp;
	_rtrigManual : R_TRIG;
	_bEnPvOld : BOOL;
	_nObjType : E_BACNETOBJECTTYPE;
END_VAR
VAR CONSTANT
	nERR_NO_ERROR		: UINT := 0;
	nERR_WRONG_MAPPING	: UINT := 2;
	nERR_OPERATIONAL	: UINT := 3;
	nERR_WRONG_TYPE		: UINT := 4;
END_VAR
(* update server device *)
IF Device._nUpdateCount = _nUpdateCount THEN
	Device();
END_IF
(* remind current number of update counter *)
_nUpdateCount := Device._nUpdateCount;

(* trigger on manual flag *)
_rtrigManual(CLK:= bManual, Q=> );

(* decode object type *)
_nObjType := F_BACnet_GetObjType(_ObjectId);

(* check BitString format of StatusFlags --> if StatusFlags are less than 4, object isn't linked correctly *)
IF _nObjType <> BACnetObjectType_AnalogValue THEN
	(* wrong mapped object type *)
	nErrorId := nERR_WRONG_TYPE;
	bReady := FALSE;
	bPvDone := FALSE;

ELSIF (_StatusFlags < 4) THEN
	(* wrong mapping *)
	nErrorId := nERR_WRONG_MAPPING;
	bReady := FALSE;
	bPvDone := FALSE;

ELSIF Device.bOperational THEN
	(* write present_value on manual trigger, on-change and on operational recover *)
	IF		_rtrigManual.Q
		OR	((NOT F_BACnet_RealEQ(fPV, _PresentValue_Ads)) AND bEnablePV)
		OR	((NOT bReady) AND bManual)
		OR	(bEnablePV <> _bEnPvOld)
	THEN
		_WriteProp.bExecute := TRUE;
		bPvDone := FALSE;
		(* write depending on enable state *)
		IF bEnablePV THEN
			_PresentValue_Ads := fPV;
		ELSE
			_PresentValue_Ads := F_BACnet_NAN();
		END_IF
		_bEnPvOld := bEnablePV;
	END_IF

	(* ready state *)
	bReady := TRUE;
	nErrorId := nERR_NO_ERROR;

	(* present value *)
	fPresentValue := _PresentValue;

	(* build bit states *)
	_StatusFlagsBits := F_BACnet_StatusFlags(_StatusFlags);

	(* copy states to output *)
	bOverridden := _StatusFlagsBits.overridden;
	bOutOfService := _StatusFlagsBits.out_of_service;
	bFault := _StatusFlagsBits.fault;
	bInAlarm := _StatusFlagsBits.in_alarm;

ELSIF Device.bFirstCycle THEN
	(* first call of the server device since reboot/reset *)
	bReady := FALSE;
	bPvDone := FALSE;
ELSE
	(* server device not ready, reset local ready also *)
	bReady := FALSE;
	nErrorId := nERR_OPERATIONAL;
	bPvDone := FALSE;
END_IF

(* call write property command *)
_WriteProp(
	BACnetDevicePort	:= Device.nAdsPort,
	bExecute			:= ,
	sNetId				:= Device.sAmsNetId,
	ObjectType			:= _nObjType,
	PropertyID			:= BACnetPropertyIdentifier_PresentValue,
	Priority			:= ePriority,
	DataType			:= BACnetDataType_Real,
	ObjectInstance		:= F_BACnet_GetObjInstance(_ObjectId),
	ptrValue			:= ADR(_PresentValue_Ads),
	nLenValue			:= SIZEOF(_PresentValue_Ads),
	bDone				=> ,
	bBusy				=> ,
	bError				=> ,
	nErrID				=> nAdsErrorId);

(* set done flag *)
IF _WriteProp.bExecute AND (NOT _WriteProp.bBusy) THEN
	(* reset execution bit *)
	_WriteProp(bExecute := FALSE);
	(* check if command was finished with error *)
	IF _WriteProp.bError THEN
		IF bManual THEN
			(* retrigger if manual flag is set *)
			_WriteProp.bExecute := TRUE;
		END_IF
		bPvDone := FALSE;
	ELSE
		(* successful written *)
		bPvDone	:= TRUE;
	END_IF
END_IF

(* set error flag *)
bError := (nErrorId <> nERR_NO_ERROR) OR (nAdsErrorId <> 0);
END_FUNCTION_BLOCK

(* POU FB_BACnet_AnalogValue_EX, ST *)
FUNCTION_BLOCK FB_BACnet_AnalogValue_EX
VAR_INPUT
	bEnablePV		: BOOL; (* enable present value with priority x in priority array, FALSE = priority x disable *)
	fPV		: REAL; (* decimal number for priority x, when input bEnablePV is TRUE *)
END_VAR
VAR_IN_OUT
	Device	: FB_BACnet_Device;
END_VAR
VAR_OUTPUT
	bReady			: BOOL;
	fPresentValue	: REAL;
	bOverridden		: BOOL;
	bOutOfService	: BOOL;
	bFault			: BOOL;
	bInAlarm		: BOOL;
	bOverRange		: BOOL;
	bUnderRange		: BOOL;
	bOtherFault		: BOOL;
	eEventState		: E_BACNETEVENTSTATE;
	bAckedTrans_ToOffNormal : BOOL;
	bAckedTrans_ToFault		: BOOL;
	bAckedTrans_ToNormal	: BOOL;
	nActivePrio		: UINT;
	bError			: BOOL;
	nErrorId		: UINT;
END_VAR
VAR
	_PresentValue AT%I*: REAL; 			(* ~(BACnet_PresentValue 				:		: )
								   			(BACnet_ObjectType 					: AV	: )	*)
    _PresentValue_Priority12 AT%Q*: REAL;(* ~(BACnet_PresentValue_Priority12		:		: )	*)
	_StatusFlags AT%I*: WORD; 			(* ~(BACnet_StatusFlags 				:		: )	*)
	_StatusFlagsBits : ST_BACnet_StatusFlags;
	_EventState AT%I*: WORD;			(* ~(BACnet_EventState 					:		: )	*)
	_Reliability AT%I*: WORD;			(* ~(BACnet_Reliability 				:		: )	*)
	_ActivePriority AT%I*: UDINT; 		(* ~(BACnet_ActivePriority 				:		: )	*)
	_AckedTransitions AT%I*:WORD;		(* ~(BACnet_AckedTransitions:		: ) *)
	_AckedTransBits : ST_BACnet_EventTransitionBits;
	_nUpdateCount : UDINT := 0;
END_VAR
VAR CONSTANT
	nERR_NO_ERROR		: UINT := 0;
	nERR_WRONG_MAPPING	: UINT := 2;
	nERR_OPERATIONAL	: UINT := 3;
END_VAR
(* update server device *)
IF Device._nUpdateCount = _nUpdateCount THEN
	Device();
END_IF
(* remind current number of update counter *)
_nUpdateCount := Device._nUpdateCount;

(* check BitString format of StatusFlags --> if StatusFlags are less than 4, object isn't linked correctly *)
IF (_StatusFlags < 4) OR _AckedTransitions < 5 THEN
	(* wrong mapping *)
	nErrorId := nERR_WRONG_MAPPING;
	bReady := FALSE;

ELSIF Device.bOperational THEN
	(* ready state *)
	bReady := TRUE;
	nErrorId := nERR_NO_ERROR;

	(* write into priority array *)
	IF bEnablePV THEN
		_PresentValue_Priority12	:= fPV;
	ELSE
		_PresentValue_Priority12	:= F_BACnet_NAN();
	END_IF

	(* present value *)
	fPresentValue := _PresentValue;

	(* build bit states *)
	_StatusFlagsBits := F_BACnet_StatusFlags(_StatusFlags);
	_AckedTransBits		:= F_BACnet_EventTransitionFlags(_AckedTransitions);

	(* copy states to output *)
	bOverridden := _StatusFlagsBits.overridden;
	bOutOfService := _StatusFlagsBits.out_of_service;
	bFault := _StatusFlagsBits.fault;
	bInAlarm := _StatusFlagsBits.in_alarm;
	bOverRange := (_Reliability = BACnetReliability_over_range);
	bUnderRange := (_Reliability = BACnetReliability_under_range);
	bOtherFault := (_Reliability = BACnetReliability_unreliable_other);
	bAckedTrans_ToOffNormal := _AckedTransBits.to_offnormal;
	bAckedTrans_ToFault := _AckedTransBits.to_fault;
	bAckedTrans_ToNormal := _AckedTransBits.to_normal;

	(* convert enumeration *)
	eEventState := _EventState;

	(* copy active priority *)
	nActivePrio := UDINT_TO_UINT(_ActivePriority);
ELSIF Device.bFirstCycle THEN
	(* first call of the server device since reboot/reset *)
	bReady := FALSE;
	_PresentValue_Priority12 := F_BACnet_NAN();
ELSE
	(* server device not ready, reset local ready also *)
	bReady := FALSE;
	nErrorId := nERR_OPERATIONAL;
END_IF
(* set error flag *)
bError := (nErrorId <> nERR_NO_ERROR);
END_FUNCTION_BLOCK

(* POU FB_BACnet_BinaryInput, ST *)
FUNCTION_BLOCK FB_BACnet_BinaryInput
VAR_IN_OUT
	Device	: FB_BACnet_Device;
END_VAR
VAR_OUTPUT
	bReady			: BOOL;
	bPresentValue	: BOOL;
	bOverridden		: BOOL;
	bOutOfService	: BOOL;
	bFault			: BOOL;
	bInAlarm		: BOOL;
	bError			: BOOL;
	nErrorId		: UINT;
END_VAR
VAR
	_PresentValue AT%I*: WORD; 				(* ~(BACnet_PresentValue 		:		: )
												(BACnet_ObjectType			:BI    	: )	*)
	_StatusFlags AT%I*: WORD; 				(* ~(BACnet_StatusFlags 		:	    : )	*)
	_StatusFlagsBits : ST_BACnet_StatusFlags;
	_nUpdateCount : UDINT := 0;
END_VAR
VAR CONSTANT
	nERR_NO_ERROR		: UINT := 0;
	nERR_WRONG_MAPPING	: UINT := 2;
	nERR_OPERATIONAL	: UINT := 3;
END_VAR
(* update server device *)
IF Device._nUpdateCount = _nUpdateCount THEN
	Device();
END_IF
(* remind current number of update counter *)
_nUpdateCount := Device._nUpdateCount;

(* check BitString format of StatusFlags --> if StatusFlags are less than 4, object isn't linked correctly *)
IF (_StatusFlags < 4) THEN
	(* wrong mapping *)
	nErrorId := nERR_WRONG_MAPPING;
	bReady := FALSE;

ELSIF Device.bOperational THEN
	(* ready state *)
	bReady := TRUE;
	nErrorId := nERR_NO_ERROR;

	(* present value *)
	bPresentValue := F_BinPV_To_Bool(_PresentValue);

	(* build bit states *)
	_StatusFlagsBits := F_BACnet_StatusFlags(_StatusFlags);

	(* copy states to output *)
	bOverridden := _StatusFlagsBits.overridden;
	bOutOfService := _StatusFlagsBits.out_of_service;
	bFault := _StatusFlagsBits.fault;
	bInAlarm := _StatusFlagsBits.in_alarm;

ELSE
	bReady := FALSE;
	nErrorId := nERR_OPERATIONAL;
END_IF
(* set error flag *)
bError := (nErrorId <> nERR_NO_ERROR);
END_FUNCTION_BLOCK

(* POU FB_BACnet_BinaryInput_EX, ST *)
FUNCTION_BLOCK FB_BACnet_BinaryInput_EX
VAR_IN_OUT
	Device	: FB_BACnet_Device;
END_VAR
VAR_OUTPUT
	bReady			: BOOL;
	bPresentValue	: BOOL;
	bOverridden		: BOOL;
	bOutOfService	: BOOL;
	bFault			: BOOL;
	bInAlarm		: BOOL;
	bNoSensor		: BOOL;
	bOpenLoop		: BOOL;
	bShortedLoop	: BOOL;
	bOtherFault		: BOOL;
	eEventState		: E_BACNETEVENTSTATE;
	bAckedTrans_ToOffNormal : BOOL;
	bAckedTrans_ToFault		: BOOL;
	bAckedTrans_ToNormal	: BOOL;
	bError			: BOOL;
	nErrorId		: UINT;
END_VAR
VAR
	_PresentValue AT%I*: WORD; 				(* ~(BACnet_PresentValue 		:		: )
												(BACnet_ObjectType			:BI    	: )	*)
	_StatusFlags AT%I*: WORD; 				(* ~(BACnet_StatusFlags 		:	    : )	*)
	_StatusFlagsBits : ST_BACnet_StatusFlags;
	_EventState AT%I*: WORD; 				(* ~(BACnet_EventState 			:	    : )	*)
	_Reliability AT%I*: WORD; 				(* ~(BACnet_Reliability 		:		: )	*)
	_AckedTransitions AT%I*:WORD;			(* ~(BACnet_AckedTransitions:		: ) *)
	_AckedTransBits : ST_BACnet_EventTransitionBits;
	_nUpdateCount : UDINT := 0;
END_VAR
VAR CONSTANT
	nERR_NO_ERROR		: UINT := 0;
	nERR_WRONG_MAPPING	: UINT := 2;
	nERR_OPERATIONAL	: UINT := 3;
END_VAR
(* update server device *)
IF Device._nUpdateCount = _nUpdateCount THEN
	Device();
END_IF
(* remind current number of update counter *)
_nUpdateCount := Device._nUpdateCount;

(* check BitString format of StatusFlags --> if StatusFlags are less than 4, object isn't linked correctly *)
IF (_StatusFlags < 4) OR _AckedTransitions < 5 THEN
	(* wrong mapping *)
	nErrorId := nERR_WRONG_MAPPING;
	bReady := FALSE;

ELSIF Device.bOperational THEN
	(* ready state *)
	bReady := TRUE;
	nErrorId := nERR_NO_ERROR;

	(* present value *)
	bPresentValue := F_BinPV_To_Bool(_PresentValue);

	(* build bit states *)
	_StatusFlagsBits := F_BACnet_StatusFlags(_StatusFlags);
	_AckedTransBits		:= F_BACnet_EventTransitionFlags(_AckedTransitions);

	(* copy states to output *)
	bOverridden := _StatusFlagsBits.overridden;
	bOutOfService := _StatusFlagsBits.out_of_service;
	bFault := _StatusFlagsBits.fault;
	bInAlarm := _StatusFlagsBits.in_alarm;
	bNoSensor := (_Reliability = BACnetReliability_no_sensor);
	bOpenLoop := (_Reliability = BACnetReliability_open_loop);
	bShortedLoop := (_Reliability = BACnetReliability_shorted_loop);
	bOtherFault := (_Reliability = BACnetReliability_unreliable_other);
	bAckedTrans_ToOffNormal := _AckedTransBits.to_offnormal;
	bAckedTrans_ToFault := _AckedTransBits.to_fault;
	bAckedTrans_ToNormal := _AckedTransBits.to_normal;

	(* convert enumeration *)
	eEventState := _EventState;

ELSE
	bReady := FALSE;
	nErrorId := nERR_OPERATIONAL;
END_IF
(* set error flag *)
bError := (nErrorId <> nERR_NO_ERROR);
END_FUNCTION_BLOCK

(* POU FB_BACnet_BinaryInput_RAW, ST *)
FUNCTION_BLOCK FB_BACnet_BinaryInput_RAW
VAR_INPUT
	bRawIn			AT%Q*: BOOL;(* ~(BACnet_RawIoBinaryBoolValue : : ) *)
END_VAR
VAR_IN_OUT
	Device	: FB_BACnet_Device;
END_VAR
VAR_OUTPUT
	bReady			: BOOL;
	bPresentValue	: BOOL;
	bOverridden		: BOOL;
	bOutOfService	: BOOL;
	bFault			: BOOL;
	bInAlarm		: BOOL;
	bAckedTrans_ToOffNormal : BOOL;
	bAckedTrans_ToFault		: BOOL;
	bAckedTrans_ToNormal	: BOOL;
	bError			: BOOL;
	nErrorId		: UINT;
END_VAR
VAR
	_PresentValue AT%I*: WORD; 				(* ~(BACnet_PresentValue 		:		: )
												(BACnet_ObjectType			:BI    	: )	*)
	_StatusFlags AT%I*: WORD; 				(* ~(BACnet_StatusFlags 		:	    : )	*)
	_AckedTransitions AT%I*:WORD;			(* ~(BACnet_AckedTransitions:		: ) *)
	_AckedTransBits : ST_BACnet_EventTransitionBits;
	_StatusFlagsBits : ST_BACnet_StatusFlags;
	_nUpdateCount : UDINT := 0;
END_VAR
VAR CONSTANT
	nERR_NO_ERROR		: UINT := 0;
	nERR_WRONG_MAPPING	: UINT := 2;
	nERR_OPERATIONAL	: UINT := 3;
END_VAR
(* update server device *)
IF Device._nUpdateCount = _nUpdateCount THEN
	Device();
END_IF
(* remind current number of update counter *)
_nUpdateCount := Device._nUpdateCount;

(* check BitString format of StatusFlags --> if StatusFlags are less than 4, object isn't linked correctly *)
IF (_StatusFlags < 4) OR _AckedTransitions < 5 THEN
	(* wrong mapping *)
	nErrorId := nERR_WRONG_MAPPING;
	bReady := FALSE;

ELSIF Device.bOperational THEN
	(* ready state *)
	bReady := TRUE;
	nErrorId := nERR_NO_ERROR;

	(* present value *)
	bPresentValue := F_BinPV_To_Bool(_PresentValue);

	(* build bit states *)
	_StatusFlagsBits := F_BACnet_StatusFlags(_StatusFlags);
	_AckedTransBits		:= F_BACnet_EventTransitionFlags(_AckedTransitions);

	(* copy states to output *)
	bOverridden := _StatusFlagsBits.overridden;
	bOutOfService := _StatusFlagsBits.out_of_service;
	bFault := _StatusFlagsBits.fault;
	bInAlarm := _StatusFlagsBits.in_alarm;
	bAckedTrans_ToOffNormal := _AckedTransBits.to_offnormal;
	bAckedTrans_ToFault := _AckedTransBits.to_fault;
	bAckedTrans_ToNormal := _AckedTransBits.to_normal;

ELSE
	bReady := FALSE;
	nErrorId := nERR_OPERATIONAL;
END_IF
(* set error flag *)
bError := (nErrorId <> nERR_NO_ERROR);
END_FUNCTION_BLOCK

(* POU FB_BACnet_BinaryOutput, ST *)
FUNCTION_BLOCK FB_BACnet_BinaryOutput
VAR_INPUT
	bEnablePV	: BOOL; (* enable present value with priority x in priority array, FALSE = priority x disable (NULL) *)
	bPV			: BOOL; (* present value bool type *)
END_VAR
VAR_IN_OUT
	Device		: FB_BACnet_Device;
END_VAR
VAR_OUTPUT
	bReady			: BOOL;
	bPresentValue	: BOOL;
	bOverridden		: BOOL;
	bOutOfService	: BOOL;
	bFault			: BOOL;
	bInAlarm		: BOOL;
	bError			: BOOL;
	nErrorId		: UINT;
END_VAR
VAR
	_PresentValue AT%I*: WORD; 			(* ~(BACnet_PresentValue 			:		: )
								   			(BACnet_ObjectType 				: BO	: )	*)
    _PresentValue_Priority12 AT%Q*: WORD;(* ~(BACnet_PresentValue_Priority12	:		: )	*)
	_StatusFlags AT%I*: WORD; 			(* ~(BACnet_StatusFlags 			:		: )	*)
	_StatusFlagsBits : ST_BACnet_StatusFlags;
	_nUpdateCount : UDINT := 0;
END_VAR
VAR CONSTANT
	nERR_NO_ERROR		: UINT := 0;
	nERR_WRONG_MAPPING	: UINT := 2;
	nERR_OPERATIONAL	: UINT := 3;
END_VAR
(* update server device *)
IF Device._nUpdateCount = _nUpdateCount THEN
	Device();
END_IF
(* remind current number of update counter *)
_nUpdateCount := Device._nUpdateCount;

(* check BitString format of StatusFlags --> if StatusFlags are less than 4, object isn't linked correctly *)
IF (_StatusFlags < 4) THEN
	(* wrong mapping *)
	nErrorId := nERR_WRONG_MAPPING;
	bReady := FALSE;

ELSIF Device.bOperational THEN
	(* ready state *)
	bReady := TRUE;
	nErrorId := nERR_NO_ERROR;

	(* write into priority array *)
	_PresentValue_Priority12 := F_Bool_To_BinPV(bEnablePV, bPV);

	(* present value *)
	bPresentValue := F_BinPV_To_Bool(_PresentValue);

	(* build bit states *)
	_StatusFlagsBits := F_BACnet_StatusFlags(_StatusFlags);

	(* copy states to output *)
	bOverridden := _StatusFlagsBits.overridden;
	bOutOfService := _StatusFlagsBits.out_of_service;
	bFault := _StatusFlagsBits.fault;
	bInAlarm := _StatusFlagsBits.in_alarm;

